expect(condition := rejected, message := 'Recovery rejects missing storage before any child access');
expectDInt(
	expected := -1,
	actual := _MissingConfigurationRunner.ExitCode,
	message := 'Invalid recovery retains abort'
);
rejected := FALSE;

__TRY
	_ExceptionAdsReporter.ReportTestCaseResult(
		groupPath := "",
		testName := "Invalid ADS outcome",
		outcome := TOF_Testing.TEST_OUTCOME.RUNNING,
		duration := T#0S,
		message := diagnostic
	);
__CATCH(exceptionCode)
	assertCaughtExceptionType(exceptionCode := exceptionCode, expectedTypeName := 'ArgumentValueNotSupportedException');
	rejected := TRUE;
__ENDTRY

expect(condition := rejected, message := 'Reporter rejects the actual nonterminal enum value');
checkExceptionClasses := TRUE;
END_METHOD

(*!
<summary>Verifies first-failure summary retention and per-run reset through the ADS reporter callbacks.</summary>
<description>Checks rejected writes, bounded ADS output for a root leaf, and reset on the next run.
Returns TRUE when all observations for this scenario are complete.
</description>
*)
METHOD PRIVATE checkAdsReporterSummary : BOOL
VAR
	diagnostic : TOF_Core.ERROR_MESSAGE;
END_VAR
_AdsSummaryReporter.ReportRunStart(testCount := 2);
_AdsSummaryReporter.RejectWrites := TRUE;
diagnostic := "Synthetic first diagnostic";
_AdsSummaryReporter.ReportTestCaseResult(
	groupPath := "Reporter regression",
	testName := "First leaf",
	outcome := TOF_Testing.TEST_OUTCOME.FAILED,
	duration := T#0S,
	message := diagnostic
);

_AdsSummaryReporter.RejectWrites := FALSE;
diagnostic := "Synthetic second diagnostic";
_AdsSummaryReporter.ReportTestCaseResult(
	groupPath := "Reporter regression",
	testName := "Second leaf",
	outcome := TOF_Testing.TEST_OUTCOME.FAILED,
	duration := T#0S,
	message := diagnostic
);

_AdsSummaryReporter.ReportRunEnd(
	totalTests := 2,
	passedTests := 0,
	failedTests := 2,
	skippedTests := 0,
	duration := T#0S
);

expect(
	condition := _AdsSummaryReporter.LastRunSummary =
		"[TOF_Testing] Finished: 0 passed, 2 failed, 0 skipped | First failure: First leaf: Synthetic first diagnostic",
	message := 'A second failure must preserve the first failure in the summary'
);

expect(
	condition := _AdsSummaryReporter.AcceptedMessage =
		"[TOF_Testing] Finished: 0 passed, 2 failed, 0 skipped | First failed test: First leaf",
	message := 'The completion record must identify the first failure even after its detail write is rejected'
);
expect(
	condition := _AdsSummaryReporter.FailedLogWriteCount = 1,
	message := 'Exactly one rejected write must be counted'
);
expect(
	condition := _AdsSummaryReporter.LastLogFailureMessage =
		"[TOF_Testing] Reporter regression/First leaf: Synthetic first diagnostic",
	message := 'Later accepted writes must preserve the rejected message'
);

_AdsSummaryReporter.ReportRunStart(testCount := 0);

expect(
	condition := _AdsSummaryReporter.LastRunSummary = "",
	message := 'Starting a new run must clear the retained summary'
);
expect(
	condition := _AdsSummaryReporter.FailedLogWriteCount = 0 AND_THEN _AdsSummaryReporter.LastLogFailureMessage = "",
	message := 'A successful start must clear earlier failed-write observations'
);

_AdsSummaryReporter.ReportRunEnd(
	totalTests := 0,
	passedTests := 0,
	failedTests := 0,
	skippedTests := 0,
	duration := T#0S
);

expect(
	condition := _AdsSummaryReporter.LastRunSummary = "[TOF_Testing] Finished: 0 passed, 0 failed, 0 skipped",
	message := 'An empty run must omit the earlier failure'
);

_AdsSummaryReporter.ReportRunStart(testCount := 1);
diagnostic := "Long diagnostic containing a literal %s. ";
TOF_Core.WideStrings.AppendFit255(
	diagnostic,
	"AAAAAAAAAAAAAAAAAAAAAAAAAAAAAAAAAAAAAAAAAAAAAAAAAAAAAAAAAAAAAAAAAAAAAAAAAAAAAAAA",
	"BBBBBBBBBBBBBBBBBBBBBBBBBBBBBBBBBBBBBBBBBBBBBBBBBBBBBBBBBBBBBBBBBBBBBBBBBBBBBBBB",
	"CCCCCCCCCCCCCCCCCCCCCCCCCCCCCCCCCCCCCCCCCCCCCCCCCCCCCCCCCCCCCCCCCCCCCCCCCCCCCCCC"
);
_AdsSummaryReporter.ReportTestCaseResult(
	groupPath := "",
	testName := "Long failure",
	outcome := TOF_Testing.TEST_OUTCOME.FAILED,
	duration := T#0S,
	message := diagnostic
);

expect(
	condition := TOF_Core.WideStrings.GetLength(value := _AdsSummaryReporter.AcceptedMessage) = 200,
	message := 'A long ADS diagnostic must fit within the reporter limit'
);
expect(
	condition := Tc2_Standard.WLEFT(STR := _AdsSummaryReporter.AcceptedMessage, SIZE := 27) =
		"[TOF_Testing] Long failure:",
	message := 'A root leaf is logged without a leading group separator'
);

_AdsSummaryReporter.RejectWrites := TRUE;
_AdsSummaryReporter.ReportRunEnd(
	totalTests := 1,
	passedTests := 0,
	failedTests := 1,
	skippedTests := 0,
	duration := T#0S
);
expect(
	condition := _AdsSummaryReporter.LastLogFailureMessage =
		"[TOF_Testing] Finished: 0 passed, 1 failed, 0 skipped | First failed test: Long failure",
	message := 'Rejection must retain the exact completion record independently of diagnostic length'
);
expect(
	condition := _AdsSummaryReporter.FailedLogWriteCount = 1,
	message := 'A rejected completion record must be counted once'
);
_AdsSummaryReporter.RejectWrites := FALSE;

checkAdsReporterSummary := TRUE;
END_METHOD

(*!
<summary>Recovers a throwing external child, including a failed first recovery attempt.</summary>
<description>Explicitly releases the modeled resource before requesting reset recovery.
Returns TRUE when all observations for this scenario are complete.
</description>
*)
METHOD PRIVATE checkExternalRecovery : BOOL
VAR
	exceptionCode : __SYSTEM.ExceptionCode;
	rejected : BOOL;
	externalCase : REFERENCE TO ExternalElementProbe;
	actualParent : TOF_Testing.ITestElement;
END_VAR
IF NOT _ExternalConfigured THEN
	_ExternalRun.Reporter := _ExternalReport;
	_ExternalConfigured := TRUE;
END_IF

_ExternalRun.Execute(cleanupTaskMemory := FALSE);
_ExternalCalls := _ExternalCalls + 1;

IF NOT _ExternalRun.IsFinished THEN
	IF _ExternalCalls < 16 THEN
		RETURN;
	END_IF

	expect(condition := FALSE, message := 'The external recovery run must finish within 16 scans');
	_ExternalRun.ExternalCase.ReleaseResource();
	checkExternalRecovery := TRUE;

	RETURN;
END_IF

IF NOT _ExternalRecovered THEN
	expectDInt(expected := -1, actual := _ExternalRun.ExitCode, message := 'External child aborts');
	expect(
		condition := _ExternalRun.ExternalCase.ResourceActive,
		message := 'Abort does not silently release user resources'
	);
	_ExternalRun.Execute(cleanupTaskMemory := FALSE);
	expectUDInt(
		expected := 1,
		actual := _ExternalRun.ExternalCase.ExecuteCalls,
		message := 'The aborted callback is not retried before explicit recovery'
	);
	externalCase REF= _ExternalRun.ExternalCase;
	externalCase.ReleaseResource();
	expectFalse(
		condition := externalCase.ResourceActive,
		message := 'Explicit resource release completes before reset recovery'
	);
	externalCase.ThrowOnReset := TRUE;

	__TRY
		_ExternalRun.Reset();
	__CATCH(exceptionCode)
		assertCaughtExceptionType(
			exceptionCode := exceptionCode,
			expectedTypeName := 'StandardException'
		);
		rejected := TRUE;
	__ENDTRY

	expect(condition := rejected, message := 'Custom recovery Reset failure propagates');
	expectDInt(expected := -1, actual := _ExternalRun.ExitCode, message := 'Failed recovery retains abort');
	externalCase.ThrowOnReset := FALSE;
	externalCase.ThrowOnExecute := FALSE;
	_ExternalRun.Reset();
	actualParent := _ExternalRun.ExternalCase.Parent;
	expect(condition := actualParent = 0, message := 'The recovered root remains parentless');
	expectUDInt(
		expected := 3,
		actual := _ExternalRun.ExternalCase.ResetCalls,
		message := 'Failed reset was retried'
	);
	_ExternalRecovered := TRUE;
	_ExternalCalls := 0;
	RETURN;
END_IF

expect(condition := _ExternalRun.AllPassed, message := 'The same static tree succeeds after explicit recovery');
expectDInt(expected := 1, actual := _ExternalRun.PassedTests, message := 'The recovered root contributes one leaf');
expect(condition := _ExternalReport.IsReady, message := 'The recovered run completes its report');
expectUDInt(
	expected := 2,
	actual := _ExternalRun.ExternalCase.ExecuteCalls,
	message := 'Execute resumes only in the new run'
);
checkExternalRecovery := TRUE;
END_METHOD

(*!
<summary>Checks direct-child interface dispatch, fixed ordering and explicit accessor failures.</summary>
<description>
Borrows persistent fixtures before execution and after a rejected Reset. Test-only slot corruption is restored
before returning. Child identity is compared through ITestElement on both sides; indexed observation
invokes no child body.

Returns TRUE when all observations for this scenario are complete.
</description>
*)
METHOD PRIVATE checkIndexedChildren : BOOL
VAR
	element : TOF_Testing.ITestElement;
	parentElement : TOF_Testing.IParentTestElement;
	child : TOF_Testing.ITestElement;
	expectedChild : TOF_Testing.ITestElement;
	supportsChildren : BOOL;
	exceptionCode : __SYSTEM.ExceptionCode;
	rejected : BOOL;
	firstBodyCalls : UDINT;
END_VAR
element := _IndexedGroup;
supportsChildren := __QUERYINTERFACE(element, parentElement);
expect(condition := supportsChildren, message := 'A group exposes the direct-child capability');

IF NOT supportsChildren THEN
	checkIndexedChildren := TRUE;
	RETURN;
END_IF

firstBodyCalls := _IndexedGroup.First.BodyCalls;
expect(condition := parentElement.ChildCount = 2, message := 'The capability reports the fixed direct count');
expectedChild := _IndexedGroup.First;
child := parentElement.GetChildByIndex(index := 0);
expect(condition := child = expectedChild, message := 'Index zero borrows the first child');
expectedChild := _IndexedGroup.Second;
child := parentElement.GetChildByIndex(index := 1);
expect(condition := child = expectedChild, message := 'The last valid index borrows the last child');

__TRY
	child := parentElement.GetChildByIndex(index := 2);
__CATCH(exceptionCode)
	assertCaughtExceptionType(exceptionCode := exceptionCode, expectedTypeName := 'ArgumentOutOfRangeException');
	rejected := TRUE;
__ENDTRY

expect(condition := rejected, message := 'Index equal to ChildCount is rejected');
rejected := FALSE;

__TRY
	child := parentElement.GetChildByIndex(index := TOF_Core.SignedInt16.MAX_VALUE);
__CATCH(exceptionCode)
	assertCaughtExceptionType(exceptionCode := exceptionCode, expectedTypeName := 'ArgumentOutOfRangeException');
	rejected := TRUE;
__ENDTRY

expect(condition := rejected, message := 'The largest representable index is rejected before indexing');
parentElement := _Runner.Empty;
expect(condition := parentElement.ChildCount = TOF_Core.SignedInt16.ZERO, message := 'An empty group reports zero direct children');
rejected := FALSE;

__TRY
	child := parentElement.GetChildByIndex(index := 0);
__CATCH(exceptionCode)
	assertCaughtExceptionType(exceptionCode := exceptionCode, expectedTypeName := 'ArgumentOutOfRangeException');
	rejected := TRUE;
__ENDTRY

expect(condition := rejected, message := 'A valid empty array has no valid child index');
parentElement := _MissingConfigurationGroup;
rejected := FALSE;

__TRY
	child := parentElement.GetChildByIndex(index := TOF_Core.SignedInt16.MAX_VALUE);
__CATCH(exceptionCode)
	assertCaughtExceptionType(exceptionCode := exceptionCode, expectedTypeName := 'DataMemberNotSpecifiedException');
	rejected := TRUE;
__ENDTRY

expect(condition := rejected, message := 'Missing storage is diagnosed before an invalid index');

// A failed Reset does not prevent observing an existing slot; the missing selected slot remains an error.
_IndexedGroup.Children[1] := 0;
rejected := FALSE;

__TRY
	_IndexedGroup.Reset(reporter := 0);
__CATCH(exceptionCode)
	assertCaughtExceptionType(exceptionCode := exceptionCode, expectedTypeName := 'DataMemberNotSpecifiedException');
	rejected := TRUE;
__ENDTRY

expect(condition := rejected, message := 'The injected missing slot rejects Reset');
parentElement := _IndexedGroup;
expectedChild := _IndexedGroup.First;
child := parentElement.GetChildByIndex(index := 0);
expect(condition := child = expectedChild, message := 'An existing slot can be observed after failed Reset');
rejected := FALSE;

__TRY
	child := parentElement.GetChildByIndex(index := 1);
__CATCH(exceptionCode)
	assertCaughtExceptionType(exceptionCode := exceptionCode, expectedTypeName := 'DataMemberNotSpecifiedException');
	rejected := TRUE;
__ENDTRY

expect(condition := rejected, message := 'A null selected slot is a missing member');
_IndexedGroup.Children[1] := _IndexedGroup.Second;
expectUDInt(
	expected := firstBodyCalls,
	actual := _IndexedGroup.First.BodyCalls,
	message := 'Indexed observation invokes no child body'
);
_IndexedGroup.Reset(reporter := 0);
checkIndexedChildren := TRUE;
END_METHOD

(*!
<summary>Checks live root-to-element paths independently of Reset and reporting.</summary>
<description>
Checks interface dispatch, own-name inclusion, empty names, Unicode, root-prefix truncation and cycles among ancestors.
Synthetic parent-only chains isolate GetPath; they are never registered or executed as group compositions.
The existing nested and repeated-run cases independently check JUnit group paths without the leaf name.

Returns TRUE when all observations for this scenario are complete.
</description>
*)
METHOD PRIVATE checkPaths : BOOL
VAR
	element : TOF_Testing.ITestElement;
	named : TOF_Core.INamed;
	actualPath : WSTRING(255);
	expectedPath : WSTRING(255);
	exceptionCode : __SYSTEM.ExceptionCode;
	rejected : BOOL;
	diagnostic : TOF_Core.ERROR_MESSAGE;
	content : POINTER TO STRING;
	longName : WSTRING(81);
	expectedXmlName : STRING(255);
END_VAR
expectedPath := "AAAAAAAAAAAAAAAAAAAAAAAAAAAAAAAAAAAAAAAAAAAAAAAAAAAAAAAAAAAAAAAAAAAAAAAAAAAAAAAA";
named := _PathLongName;
expect(condition := named.Name = expectedPath, message := 'INamed retains the first 80 name characters');
actualPath := _PathLongName.GetPath();
expect(condition := actualPath = expectedPath, message := 'A root path observes the same bounded name');
longName := "AAAAAAAAAAAAAAAAAAAAAAAAAAAAAAAAAAAAAAAAAAAAAAAAAAAAAAAAAAAAAAAAAAAAAAAAAAAAAAAAB";
_PathReport.ReportRunStart(testCount := 1);
_PathReport.ReportTestCaseResult(
	groupPath := "",
	testName := longName,
	outcome := TOF_Testing.TEST_OUTCOME.PASSED,
	duration := T#0S,
	message := diagnostic
);
_PathReport.ReportRunEnd(totalTests := 1, passedTests := 1, failedTests := 0, skippedTests := 0, duration := T#0S);
content := _PathReport.ContentAddress;
expectedXmlName := TOF_Core.Strings.Concat255('name="', TO_STRING(expectedPath), '"');
expect(condition := _PathReport.IsReady AND_THEN content <> 0, message := 'The bounded-name report completes');

IF content <> 0 THEN
	expect(
		condition := TOF_Core.Strings.Contains(stringToSearchIn := content^, stringToFind := expectedXmlName),
		message := 'Reporter input retains exactly the first 80 name characters'
	);
END_IF

element := _DuplicateGroup;
actualPath := element.GetPath();
expect(condition := actualPath = "Duplicates", message := 'A root path contains its own name');
actualPath := _DuplicateGroup.First.GetPath();
expect(condition := actualPath = "Duplicates/First", message := 'A child path includes its group and own name');
actualPath := _Runner.FailureOuter.Failures.BodyFailure.GetPath();
expect(
	condition := actualPath = "Nested/Failures/Body failure",
	message := 'Ancestor names are ordered from the root'
);
actualPath := _Runner.Pass.GetPath();
expect(condition := actualPath = "", message := 'A nameless root has an empty path');
actualPath := _PathEmpty.GetPath();
expectedPath := "AAAAAAAAAAAAAAAAAAAAAAAAAAAAAAAAAAAAAAAAAAAAAAAAAAAAAAAAAAAAAAAAAAAAAAAAAAAAAAAA";
expect(condition := actualPath = expectedPath, message := 'An empty own name adds no separator');
actualPath := _PathUnicode.GetPath();
expectedPath := "AAAAAAAAAAAAAAAAAAAAAAAAAAAAAAAAAAAAAAAAAAAAAAAAAAAAAAAAAAAAAAAAAAAAAAAAAAAAAAAA/Ω";
expect(condition := actualPath = expectedPath, message := 'Empty ancestors are skipped and Unicode is preserved');
actualPath := _PathFourth.GetPath();
expectedPath := Tc2_Utilities.WCONCAT(
	STR1 := "AAAAAAAAAAAAAAAAAAAAAAAAAAAAAAAAAAAAAAAAAAAAAAAAAAAAAAAAAAAAAAAAAAAAAAAAAAAAAAAA/",
	STR2 := "BBBBBBBBBBBBBBBBBBBBBBBBBBBBBBBBBBBBBBBBBBBBBBBBBBBBBBBBBBBBBBBBBBBBBBBBBBBBBBBB/"
);
expectedPath := Tc2_Utilities.WCONCAT(
	STR1 := expectedPath,
	STR2 := "CCCCCCCCCCCCCCCCCCCCCCCCCCCCCCCCCCCCCCCCCCCCCCCCCCCCCCCCCCCCCCCCCCCCCCCCCCCCCCCC/DDDDDDDDDDD…"
);
expect(condition := actualPath = expectedPath, message := 'Overflow retains the root prefix and final ellipsis');

__TRY
	actualPath := _ParentGroup.Child.GetPath();
__CATCH(exceptionCode)
	assertCaughtExceptionType(exceptionCode := exceptionCode, expectedTypeName := 'StandardException');
	rejected := TRUE;
__ENDTRY

expect(condition := rejected, message := 'A cycle among ancestors is rejected without endless traversal');
actualPath := _ReportPathInner.GetPath();
_PathReport.ReportRunStart(testCount := 1);
_PathReport.ReportTestCaseResult(
	groupPath := actualPath,
	testName := "Leaf",
	outcome := TOF_Testing.TEST_OUTCOME.PASSED,
	duration := T#0S,
	message := diagnostic
);
_PathReport.ReportRunEnd(totalTests := 1, passedTests := 1, failedTests := 0, skippedTests := 0, duration := T#0S);
content := _PathReport.ContentAddress;
expect(condition := _PathReport.IsReady AND_THEN content <> 0, message := 'The deep-path report completes');

IF content <> 0 THEN
	expect(
		condition := TOF_Core.Strings.Contains(
			stringToSearchIn := content^,
			stringToFind := 'name="Leaf" classname="Report root/Middle/Inner"'
		),
		message := 'JUnit preserves all three group ancestors and keeps the leaf name separate'
	);
END_IF

checkPaths := TRUE;
END_METHOD

(*!
<summary>Verifies that a reporter failure aborts once after teardown and clears the reporter reference.</summary>
<description>The same leaf runs with a replacement reporter after a completed abort and Reset.
An incomplete run fails when it reaches the scan limit. Returns TRUE when the scenario has an outcome.
</description>
*)
METHOD PRIVATE checkReporterAbort : BOOL
VAR
	exceptionCode : __SYSTEM.ExceptionCode;
	rejected : BOOL;
	diagnostic : TOF_Core.ERROR_MESSAGE;
	actualParent : TOF_Testing.ITestElement;
END_VAR
IF _AbortRecovered THEN
	_AbortRun.Execute(cleanupTaskMemory := FALSE);
	_AbortCalls := _AbortCalls + 1;

	IF NOT _AbortRun.IsFinished AND_THEN _AbortCalls < 16 THEN
		RETURN;
	END_IF

	expect(condition := _AbortRun.IsFinished, message := 'The recovered reporter run finishes within 16 scans');
	expect(condition := _AbortRun.IsFinished AND_THEN _AbortRun.AllPassed,
		message := 'The same static tree passes after reporter abort');
	expectUDInt(
		expected := 1,
		actual := _AbortRun.AbortCase.BodyCalls,
		message := 'The same root executes once in the new run'
	);
	expectUDInt(expected := 1, actual := _AbortReport.ResultCalls, message := 'Old reporter is not retried');
	checkReporterAbort := TRUE;
	RETURN;
END_IF

IF NOT _AbortConfigured THEN

	__TRY
		_InvalidReport.ReportTestCaseResult(
			groupPath := "",
			testName := "Invalid outcome",
			outcome := TOF_Testing.TEST_OUTCOME.NOT_RUN,
			duration := T#0S,
			message := diagnostic
		);
	__CATCH(exceptionCode)
		assertCaughtExceptionType(
			exceptionCode := exceptionCode,
			expectedTypeName := 'ArgumentValueNotSupportedException'
		);
		rejected := TRUE;
	__ENDTRY

	expect(condition := rejected, message := 'A reporter rejects a nonterminal outcome');
	_AbortRun.Reporter := _AbortReport;
	_AbortConfigured := TRUE;
END_IF

_AbortRun.Execute(cleanupTaskMemory := FALSE);
_AbortCalls := _AbortCalls + 1;

IF NOT _AbortRun.IsFinished THEN
	IF _AbortCalls < 16 THEN
		RETURN;
	END_IF

	expect(condition := FALSE, message := 'Callback abort must terminate within 16 scans');
	checkReporterAbort := TRUE;

	RETURN;
END_IF

IF _AbortPostCalls < 2 THEN
	_AbortPostCalls := _AbortPostCalls + 1;
	RETURN;
END_IF

expectDInt(expected := -1, actual := _AbortRun.ExitCode, message := 'Callback abort has a distinct exit code');
expectUDInt(expected := 1, actual := _AbortReport.ResultCalls, message := 'The callback is never retried');
expectUDInt(
	expected := 1,
	actual := _AbortRun.AbortCase.TeardownCalls,
	message := 'Cleanup precedes result reporting'
);
expect(
	condition := _AbortRun.AbortCase.IsFinished AND_THEN _AbortRun.AbortCase.Reporter = 0,
	message := 'A completed leaf clears its reporter reference even when result delivery throws'
);
expectFalse(condition := _AbortReport.IsReady, message := 'An aborted report remains incomplete');
expect(
	condition := TOF_Core.WideStrings.Contains(stringToSearchIn := _AbortRun.CallbackMessage,
		stringToFind := "Reporter failed"),
	message := 'External callback diagnostic is copied'
);
_AbortRun.Reset();
expect(condition := _AbortRun.CallbackMessage = "", message := 'Reset clears copied callback diagnostic');
actualParent := _AbortRun.AbortCase.Parent;
expect(condition := actualParent = 0, message := 'The same root remains parentless after recovery');
_AbortRun.Reporter := _AbortRecoveryReport;
_AbortRecovered := TRUE;
_AbortCalls := 0;
END_METHOD

(*!
<summary>Checks static root validation, recovery guards and absence of cyclic topology scans.</summary>
<description>Deliberately corrupts test-only slots, restoring them before valid recovery and before execution reaches them.
Returns TRUE when all observations for this scenario are complete.
</description>
*)
METHOD PRIVATE checkRunnerTopology : BOOL
VAR
	exceptionCode : __SYSTEM.ExceptionCode;
	rejected : BOOL;
	runningRoot : REFERENCE TO AssertionIsolationProbe;
	actualParent : TOF_Testing.ITestElement;
END_VAR
IF NOT _RootTopologyConfigured THEN
	_RootTopologyRunner.Reporter := _RootTopologyReport;
	_RootTopologyRunner.RootTopologyFirst.Reset(reporter := 0);
	_RootTopologyRunner.RootTopologyFirst.Execute();
	_RootTopologyRunner.Children[1] := 0;
	_RootTopologyRunner.Execute(cleanupTaskMemory := FALSE);
	expectDInt(expected := -1, actual := _RootTopologyRunner.ExitCode, message := 'A null root aborts startup');
	assertCaughtExceptionType(
		exceptionCode := _RootTopologyRunner.CallbackException,
		expectedTypeName := 'DataMemberNotSpecifiedException'
	);
	expect(
		condition := _RootTopologyRunner.RootTopologyFirst.IsFinished,
		message := 'All direct roots are validated before the first Reset'
	);
	expectFalse(condition := _RootTopologyReport.IsReady, message := 'Invalid startup produces no completed report');
	expect(
		condition := _RootTopologyReport.ContentLength = TOF_Core.UnsignedInt32.ZERO,
		message := 'Invalid startup does not call ReportRunStart'
	);
	rejected := FALSE;

	__TRY
		_RootTopologyRunner.Reset();
	__CATCH(exceptionCode)
		assertCaughtExceptionType(exceptionCode := exceptionCode, expectedTypeName := 'DataMemberNotSpecifiedException');
		rejected := TRUE;
	__ENDTRY

	expect(condition := rejected, message := 'Recovery validates slots before dereferencing an invalid tree');
	expectDInt(
		expected := -1,
		actual := _RootTopologyRunner.ExitCode,
		message := 'Failed recovery retains abort'
	);
	_RootTopologyRunner.Children[1] := _RootTopologyRunner.RootTopologyGroup;
	_RootTopologyRunner.Reset();
	_RootTopologyRunner.Children[1] := _RootTopologyRunner.RootTopologyFirst;
	_RootTopologyRunner.Execute(cleanupTaskMemory := FALSE);
	expectDInt(
		expected := -1,
		actual := _RootTopologyRunner.ExitCode,
		message := 'Duplicate roots abort startup'
	);
	assertCaughtExceptionType(exceptionCode := _RootTopologyRunner.CallbackException, expectedTypeName := 'StandardException');
	_RootTopologyRunner.Children[1] := _RootTopologyRunner.RootTopologyGroup;
	_RootTopologyRunner.Reset();
	_RootTopologyRunner.Children[0] := _RootTopologyRunner.RootTopologyGroup.Child;
	_RootTopologyRunner.Execute(cleanupTaskMemory := FALSE);
	expectDInt(
		expected := -1,
		actual := _RootTopologyRunner.ExitCode,
		message := 'A group-owned root aborts startup'
	);
	assertCaughtExceptionType(exceptionCode := _RootTopologyRunner.CallbackException, expectedTypeName := 'StandardException');
	_RootTopologyRunner.Children[0] := _RootTopologyRunner.RootTopologyFirst;
	_RootTopologyRunner.Reset();
	_RootTopologyRunner.RootTopologyFirst.Execute();
	_RootTopologyRunner.Children[1] := _Runner.FailureOuter.Failures;
	_RootTopologyRunner.Execute(cleanupTaskMemory := FALSE);
	expectDInt(
		expected := -1,
		actual := _RootTopologyRunner.ExitCode,
		message := 'A nested group cannot also occupy a root slot'
	);
	assertCaughtExceptionType(exceptionCode := _RootTopologyRunner.CallbackException, expectedTypeName := 'StandardException');
	expect(
		condition := _RootTopologyRunner.RootTopologyFirst.IsFinished,
		message := 'Owned-group rejection occurs before the first direct Reset'
	);
	expect(
		condition := _RootTopologyReport.ContentLength = TOF_Core.UnsignedInt32.ZERO,
		message := 'Owned-group rejection does not start reporting'
	);
	rejected := FALSE;

	__TRY
		_RootTopologyRunner.Reset();
	__CATCH(exceptionCode)
		assertCaughtExceptionType(exceptionCode := exceptionCode, expectedTypeName := 'StandardException');
		rejected := TRUE;
	__ENDTRY

	expect(condition := rejected, message := 'Abort recovery also rejects a group-owned root');
	expectDInt(expected := -1, actual := _RootTopologyRunner.ExitCode, message := 'Invalid recovery retains abort');
	_RootTopologyRunner.Children[1] := _RootTopologyRunner.RootTopologyGroup;
	_RootTopologyRunner.Reset();
	runningRoot REF= _RootTopologyRunner.RunningRoot;
	runningRoot.Timeout := T#0S;
	_RootTopologyRunner.RunningRoot.Reset(reporter := 0);
	_RootTopologyRunner.RunningRoot.Execute();
	expect(condition := _RootTopologyRunner.RunningRoot.IsRunning, message := 'The active-root fixture is pending');
	_RootTopologyRunner.Children[0] := _RootTopologyRunner.RunningRoot;
	_RootTopologyRunner.Execute(cleanupTaskMemory := FALSE);
	expectDInt(
		expected := -1,
		actual := _RootTopologyRunner.ExitCode,
		message := 'An active root aborts startup'
	);
	assertCaughtExceptionType(exceptionCode := _RootTopologyRunner.CallbackException, expectedTypeName := 'StandardException');
	_RootTopologyRunner.RunningRoot.Reset(reporter := 0);
	_RootTopologyRunner.Children[0] := _RootTopologyRunner.RootTopologyFirst;
	_RootTopologyRunner.Reset();
	_RootTopologyRunner.Execute(cleanupTaskMemory := FALSE);
	expectFalse(condition := _RootTopologyRunner.IsFinished, message := 'Valid startup prepares the static roots');

	// Fault injection: restore the unused slot immediately after driving the first root.
	_RootTopologyRunner.Children[1] := 0;
	_RootTopologyRunner.Execute(cleanupTaskMemory := FALSE);
	_RootTopologyRunner.Children[1] := _RootTopologyRunner.RootTopologyGroup;
	expectDInt(
		expected := 0,
		actual := _RootTopologyRunner.ExitCode,
		message := 'Execution does not rescan root slots'
	);
	_RootTopologyConfigured := TRUE;
END_IF

_RootTopologyRunner.Execute(cleanupTaskMemory := FALSE);
_RootTopologyCalls := _RootTopologyCalls + 1;

IF NOT _RootTopologyRunner.IsFinished AND_THEN _RootTopologyCalls < 16 THEN
	RETURN;
END_IF

expect(condition := _RootTopologyRunner.IsFinished, message := 'The topology run finishes within 16 scans');
expect(
	condition := _RootTopologyRunner.IsFinished AND_THEN _RootTopologyRunner.AllPassed,
	message := 'The owned static roots execute successfully'
);
expectDInt(
	expected := 2,
	actual := _RootTopologyRunner.PassedTests,
	message := 'Two direct or nested leaves pass'
);
expectUDInt(
	expected := 1,
	actual := _RootTopologyRunner.RootTopologyFirst.BodyCalls,
	message := 'The first root executes once in the valid run'
);
expectUDInt(
	expected := 1,
	actual := _RootTopologyRunner.RootTopologyGroup.Child.BodyCalls,
	message := 'The nested group executes its owned leaf'
);
actualParent := _RootTopologyRunner.RootTopologyFirst.Parent;
expect(condition := actualParent = 0, message := 'Runner roots remain parentless');
actualParent := _RootTopologyRunner.RootTopologyGroup.Child.Parent;
expect(
	condition := actualParent <> 0,
	message := 'A nested leaf retains its constructor-assigned parent'
);
checkRunnerTopology := TRUE;
END_METHOD

(*!
<summary>Checks fixed parents, missing or repeated children, parent mismatch, cycles, ordered dispatch and repeat execution.</summary>
<description>
Fault injection deliberately mutates a test-only array between rejected operations and briefly during execution
to detect redundant validation. Restore every unused slot before execution reaches it.

Returns TRUE when all observations for this scenario are complete.
</description>
*)
METHOD PRIVATE checkTopology : BOOL
VAR
	exceptionCode : __SYSTEM.ExceptionCode;
	rejected : BOOL;
	expectedParent : TOF_Testing.ITestElement;
	actualParent : TOF_Testing.ITestElement;
END_VAR
expectedParent := _DuplicateGroup;
actualParent := _DuplicateGroup.First.Parent;
expect(condition := actualParent = expectedParent, message := 'Parent is assigned at construction');
actualParent := _DuplicateGroup.Parent;
expect(condition := actualParent = 0, message := 'A root is constructed without a parent');

// Deliberately corrupt the borrowed test-only array to inject topology faults.
// A later execution probe restores its unused slot before that slot is reached.
_DuplicateGroup.Children[1] := 0;

__TRY
	_DuplicateGroup.Reset(reporter := 0);
__CATCH(exceptionCode)
	assertCaughtExceptionType(exceptionCode := exceptionCode, expectedTypeName := 'DataMemberNotSpecifiedException');
	rejected := TRUE;
__ENDTRY

expect(condition := rejected, message := 'A null fixed child is rejected by Reset');
expectUDInt(
	expected := 0,
	actual := _DuplicateGroup.First.BodyCalls,
	message := 'No earlier child body executes'
);
rejected := FALSE;
_DuplicateGroup.Children[1] := _DuplicateGroup.First;

__TRY
	_DuplicateGroup.Reset(reporter := 0);
__CATCH(exceptionCode)
	assertCaughtExceptionType(exceptionCode := exceptionCode, expectedTypeName := 'StandardException');
	rejected := TRUE;
__ENDTRY

expect(condition := rejected, message := 'Duplicate fixed slots are rejected');
rejected := FALSE;
_DuplicateGroup.Children[1] := _RootTopologyRunner.RootTopologyGroup.Child;

__TRY
	_DuplicateGroup.Reset(reporter := 0);
__CATCH(exceptionCode)
	assertCaughtExceptionType(exceptionCode := exceptionCode, expectedTypeName := 'StandardException');
	rejected := TRUE;
__ENDTRY

expect(condition := rejected, message := 'A child assigned to another group is rejected');
actualParent := _DuplicateGroup.First.Parent;
expect(condition := actualParent = expectedParent, message := 'Rejection never changes Parent');
_DuplicateGroup.Children[1] := _DuplicateGroup.Second;
rejected := FALSE;

__TRY
	_ParentGroup.Reset(reporter := 0);
__CATCH(exceptionCode)
	assertCaughtExceptionType(exceptionCode := exceptionCode, expectedTypeName := 'StandardException');
	rejected := TRUE;
__ENDTRY

expect(condition := rejected, message := 'A cycle assigned by constructors is rejected before recursion');

_DuplicateGroup.Reset(reporter := 0);
// Fault injection: an unused slot must not be rescanned in Execute; restore before that slot is reached.
_DuplicateGroup.Children[1] := 0;
_DuplicateGroup.Execute();
expectUDInt(
	expected := 1,
	actual := _DuplicateGroup.First.BodyCalls,
	message := 'The first Execute reaches the first owned child through Children'
);
expectUDInt(
	expected := 0,
	actual := _DuplicateGroup.Second.BodyCalls,
	message := 'The first Execute does not reach the second owned child'
);
_DuplicateGroup.Children[1] := _DuplicateGroup.Second;
_DuplicateGroup.Execute();
expect(condition := _DuplicateGroup.IsFinished, message := 'A valid static group finishes without Configure');
expectDInt(expected := 2, actual := _DuplicateGroup.PassedCount, message := 'Both owned leaves pass');
_DuplicateGroup.Reset(reporter := 0);
_DuplicateGroup.Execute();
_DuplicateGroup.Execute();
expectDInt(
	expected := 2,
	actual := _DuplicateGroup.PassedCount,
	message := 'Reset supports another fixed-tree run'
);
expectUDInt(
	expected := 1,
	actual := _DuplicateGroup.First.BodyCalls,
	message := 'A repeated leaf executes once'
);
actualParent := _DuplicateGroup.First.Parent;
expect(condition := actualParent = expectedParent, message := 'Repeated runs preserve Parent');
_DuplicateGroup.Children[1] := 0;
rejected := FALSE;

__TRY
	_DuplicateGroup.Reset(reporter := 0);
__CATCH(exceptionCode)
	assertCaughtExceptionType(exceptionCode := exceptionCode, expectedTypeName := 'DataMemberNotSpecifiedException');
	rejected := TRUE;
__ENDTRY

expect(condition := rejected, message := 'Invalid topology is rejected on a later Reset too');
expect(
	condition := _DuplicateGroup.First.IsFinished,
	message := 'Validation precedes the first direct child Reset'
);
_DuplicateGroup.Children[1] := _DuplicateGroup.Second;
checkTopology := TRUE;
END_METHOD

(*!
<summary>Checks long XML diagnostics, supplementary Unicode, isolated surrogates and XML controls.</summary>
<description>Returns TRUE when all observations for this scenario are complete.</description>
*)
METHOD PRIVATE checkXmlEncoding : BOOL
VAR
	diagnostic : TOF_Core.ERROR_MESSAGE;
	characters : POINTER TO WORD;
	content : POINTER TO STRING;
	i : UDINT;
END_VAR
// U+1F600 is a surrogate pair; it is followed by an isolated high surrogate, U+0001, TAB and ampersand.
characters := ADR(diagnostic);
characters[0] := 16#D83D;
characters[1] := 16#DE00;
characters[2] := 16#D800;
characters[3] := 16#0001;
characters[4] := 16#0009;
characters[5] := 16#0026;

FOR i := 6 TO 405 DO
	characters[i] := 16#0078;
END_FOR

characters[406] := TOF_Core.UnsignedInt16.MIN_VALUE;
TOF_Core.WideStrings.AppendFit(targetString := diagnostic, sourceString := "END_OF_XML_DIAGNOSTIC");
_XmlReport.ReportRunStart(testCount := 1);
_XmlReport.ReportTestCaseResult(
	groupPath := "Wide",
	testName := "",
	outcome := TOF_Testing.TEST_OUTCOME.FAILED,
	duration := T#1250MS,
	message := diagnostic
);
_XmlReport.ReportRunEnd(totalTests := 1, passedTests := 0, failedTests := 1, skippedTests := 0, duration := T#1250MS);
content := _XmlReport.ContentAddress;
expect(condition := _XmlReport.IsReady AND_THEN content <> 0, message := 'Completed Unicode XML has a buffer');

IF content <> 0 THEN
	expect(
		condition := TOF_Core.Strings.Contains(stringToSearchIn := content^,
			stringToFind := '&#128512;&#65533;&#65533;&#9;&amp;'),
		message := 'Surrogate pair, isolated surrogate, forbidden control and tab are encoded'
	);
	expect(
		condition := TOF_Core.Strings.Contains(stringToSearchIn := content^, stringToFind := 'END_OF_XML_DIAGNOSTIC'),
		message := 'Diagnostic suffix beyond 255 characters survives'
	);
	expect(
		condition := TOF_Core.Strings.Contains(stringToSearchIn := content^, stringToFind := 'time="1.250"'),
		message := 'JUnit duration uses decimal seconds'
	);
END_IF

checkXmlEncoding := TRUE;
END_METHOD

(*!
<summary>Repeats a nested run and checks configured and completed leaf counts, cleanup and escaped JUnit output.</summary>
<description>Configures owned fixtures through borrowed references without copying their state.
Returns TRUE when all observations for this scenario are complete.
</description>
*)
METHOD PRIVATE runAndCheck : BOOL
VAR
	content : POINTER TO STRING;
	probe : REFERENCE TO TestingProbe;
	multiCycleProbe : REFERENCE TO AssertionIsolationProbe;
END_VAR
IF NOT _Configured THEN
	expectDInt(expected := 5, actual := _Runner.FailureOuter.TestCount, message := 'Nested leaf count');
	expectDInt(expected := 0, actual := _Runner.Empty.TestCount, message := 'Empty group leaf count');
	expectDInt(expected := 1, actual := _Runner.Pass.TestCount, message := 'Single-cycle leaf count');
	expectDInt(expected := 1, actual := _Runner.Multi.TestCount, message := 'Multi-cycle leaf count');

	probe REF= _Runner.FailureOuter.Failures.SetupFailure;
	probe.ThrowBeforeTest := TRUE;
	probe REF= _Runner.FailureOuter.Failures.BodyFailure;
	probe.ThrowBody := TRUE;
	probe REF= _Runner.FailureOuter.Failures.TeardownFailure;
	probe.ThrowAfterTest := TRUE;
	probe REF= _Runner.FailureOuter.Failures.ComparisonFailure;
	probe.InvalidComparison := TRUE;
	probe REF= _Runner.FailureOuter.Failures.DiagnosticFailure;
	probe.DiagnosticFailure := TRUE;
	_Runner.Reporter := _Reporter;
	multiCycleProbe REF= _Runner.Multi;
	multiCycleProbe.Timeout := T#0S;
	_Configured := TRUE;
END_IF

_Runner.Execute(cleanupTaskMemory := FALSE);
_Calls := _Calls + 1;

IF NOT _Runner.IsFinished AND_THEN _Calls < 32 THEN
	RETURN;
END_IF

expect(condition := _Runner.IsFinished, message := 'The tree finishes within 32 scans');
expectDInt(expected := 2, actual := _Runner.PassedTests, message := 'Single and multi-cycle leaves pass');
expectDInt(expected := 5, actual := _Runner.FailedTests, message := 'Five distinct leaf failures');
expectDInt(expected := 7, actual := _Runner.TotalTests, message := 'Groups add no synthetic tests');
expectDInt(expected := 5, actual := _Runner.FailureOuter.TestCount, message := 'Leaf count survives a run');
expectUDInt(
	expected := 0,
	actual := _Runner.FailureOuter.Failures.SetupFailure.BodyCalls,
	message := 'Failed setup suppresses body'
);
expectUDInt(
	expected := 1,
	actual := _Runner.FailureOuter.Failures.SetupFailure.TeardownCalls,
	message := 'Failed setup still cleans up'
);
expectUDInt(
	expected := 1,
	actual := _Runner.FailureOuter.Failures.BodyFailure.TeardownCalls,
	message := 'Thrown body cleans up'
);
expectUDInt(
	expected := 1,
	actual := _Runner.FailureOuter.Failures.TeardownFailure.TeardownCalls,
	message := 'Thrown teardown is not retried'
);
expectUDInt(
	expected := 1,
	actual := _Runner.Pass.BodyCalls,
	message := 'Single-cycle body executes once per run'
);
expectUDInt(
	expected := 3,
	actual := _Runner.Multi.BodyCalls,
	message := 'Multi-cycle state survives three scans'
);
expectDInt(
	expected := 0,
	actual := _Runner.Empty.FailedCount,
	message := 'An empty group passes without tests'
);
expect(condition := _Reporter.IsReady, message := 'JUnit output is complete');
expect(
	condition := TOF_Core.WideStrings.Contains(stringToSearchIn := _Runner.FailureOuter.Failures.SetupFailure.FailureMessage,
		stringToFind := "BeforeTest: "),
	message := 'Preparation stage survives exception capture'
);
expect(
	condition := TOF_Core.WideStrings.Contains(stringToSearchIn := _Runner.FailureOuter.Failures.BodyFailure.FailureMessage,
		stringToFind := "Body failed"),
	message := 'Framework payload survives task cleanup'
);
expect(
	condition := TOF_Core.WideStrings.Contains(stringToSearchIn := _Runner.FailureOuter.Failures.BodyFailure.FailureMessage,
		stringToFind := "ExecuteTest"),
	message := 'Framework source survives task cleanup'
);
expect(
	condition := TOF_Core.WideStrings.Contains(stringToSearchIn := _Runner.FailureOuter.Failures.TeardownFailure.FailureMessage,
		stringToFind := "Teardown failed"),
	message := 'Teardown payload is copied'
);

content := _Reporter.ContentAddress;
expect(condition := content <> 0, message := 'Completed XML exposes a buffer');

IF content <> 0 THEN
	expect(
		condition := TOF_Core.Strings.Contains(
			stringToSearchIn := content^,
			stringToFind := 'Expected value &lt; '
		),
		message := 'An incompatible borrowed comparison remains an assertion failure'
	);
	expect(
		condition := TOF_Core.Strings.Contains(stringToSearchIn := content^, stringToFind := '&#1070;&amp;&lt;'),
		message := 'Cyrillic and XML markup are preserved'
	);
	expect(
		condition := TOF_Core.Strings.Contains(stringToSearchIn := content^, stringToFind := 'name=""'),
		message := 'Empty test name serializes safely'
	);
	expect(
		condition := TOF_Core.Strings.Contains(stringToSearchIn := content^, stringToFind := 'classname="Nested/Failures"'),
		message := 'The nested group path is preserved'
	);
END_IF

IF NOT _Repeated AND_THEN _Runner.IsFinished THEN
	_Repeated := TRUE;
	_Calls := 0;
	_Runner.Reset();
	RETURN;
END_IF

runAndCheck := TRUE;
END_METHOD

(*!
<summary>Borrows the initialized concrete class name.</summary>
*)
{attribute 'monitoring' := 'call'}
PROPERTY ClassName : REFERENCE TO STRING
GET
ClassName REF= _ClassName;
END_GET
END_PROPERTY

(*!
<summary>Borrows the project namespace name.</summary>
*)
{attribute 'monitoring' := 'call'}
PROPERTY NamespaceName : REFERENCE TO STRING
GET
NamespaceName REF= CurrentNamespace.Name;
END_GET
END_PROPERTY

END_FUNCTION_BLOCK

// ---- Tests/Testing/MixedTestRunner.TcPOU
(*
SPDX-License-Identifier: MIT
License: https://opensource.org/license/mit
*)

(*!
<summary>Runs mixed outcomes, nested groups, an empty group and a multi-cycle test.</summary>
<description>
Owns persistent root instances and fixed child storage. Use from one task without reentry.
Children borrows the same array for the instance lifetime. Root parents remain zero.
Instances must not be copied because their fixtures contain non-copyable state.
</description>
*)

{attribute 'no_assign'}
{attribute 'no_explicit_call' := 'do not call this function block directly'}
FUNCTION_BLOCK MixedTestRunner EXTENDS TOF_Testing.TestRunner<4>
VAR_STAT
	//! <summary>Class name shared by instances of this concrete runner.</summary>
	{attribute 'hide'}
	_ClassName : STRING := __POUNAME();
END_VAR
VAR_OUTPUT
	//! <summary>Owned root element used by this runner.</summary>
	FailureOuter : NestedFailureTestGroup(name := "Nested", parent := 0);
	//! <summary>Owned root element used by this runner.</summary>
	Empty : EmptyTestGroup(name := "Empty", parent := 0);
	//! <summary>Owned root element used by this runner.</summary>
	Pass : TestingProbe(name := "", parent := 0);
	//! <summary>Owned root element used by this runner.</summary>
	Multi : AssertionIsolationProbe(name := "Three cycles", parent := 0);
END_VAR
VAR
	_Children : ARRAY [0.._ChildCount - 1] OF TOF_Testing.ITestElement :=
	[
		FailureOuter,
		Pass,
		Multi,
		Empty
	];
END_VAR

(*!
<summary>Borrows the unchanged persistent root array; application code must not modify it.</summary>
*)
{attribute 'monitoring' := 'call'}
PROPERTY Children : REFERENCE TO ARRAY [0.._ChildCount - 1] OF TOF_Testing.ITestElement
GET
Children REF= _Children;
END_GET
END_PROPERTY

(*!
<summary>Borrows the concrete class name; callers must not modify the returned storage.</summary>
*)
{attribute 'monitoring' := 'call'}
PROPERTY ClassName : REFERENCE TO STRING
GET
ClassName REF= _ClassName;
END_GET
END_PROPERTY

(*!
<summary>Borrows the test project namespace; callers must not modify the returned storage.</summary>
*)
{attribute 'monitoring' := 'call'}
PROPERTY NamespaceName : REFERENCE TO STRING
GET
NamespaceName REF= CurrentNamespace.Name;
END_GET
END_PROPERTY

(*!
<summary>Reports the complete concrete instance size.</summary>
*)
{attribute 'monitoring' := 'call'}
PROPERTY SelfSize : ULINT
GET
SelfSize := XSIZEOF(THIS^);
END_GET
END_PROPERTY

END_FUNCTION_BLOCK

// ---- Tests/Testing/NestedFailureTestGroup.TcPOU
(*
SPDX-License-Identifier: MIT
License: https://opensource.org/license/mit
*)

(*!
<summary>Owns a nested group of failure scenarios.</summary>
<description>
Owns persistent child storage and fixed parent associations. Use in one task without reentry.
Children is borrowed and must not be modified by application code. Constructor callbacks are not used.
</description>
*)

{attribute 'no_assign'}
{attribute 'no_explicit_call' := 'do not call this function block directly'}
FUNCTION_BLOCK NestedFailureTestGroup EXTENDS TOF_Testing.TestGroup<1>
VAR_STAT
	//! <summary>Class name shared by all instances of this function block.</summary>
	{attribute 'hide'}
	_ClassName : STRING := __POUNAME();
END_VAR
VAR
	{attribute 'hide'}
	{attribute 'init_namespace'}
	_NamespaceName : STRING;
END_VAR
VAR_OUTPUT
	//! <summary>Owned nested failure group.</summary>
	Failures : FailureTestGroup(name := "Failures", parent := THIS^);
END_VAR
VAR
	_Children : ARRAY [0.._ChildCount - 1] OF TOF_Testing.ITestElement :=
	[
		Failures
	];
END_VAR

//! <summary>Borrows the concrete class name for the lifetime of this instance; callers must not modify it.</summary>
{attribute 'monitoring' := 'call'}
PROPERTY ClassName : REFERENCE TO STRING
GET
ClassName REF= _ClassName;
END_GET
END_PROPERTY

//! <summary>Borrows the compiler-initialized namespace; callers must not modify the returned reference.</summary>
{attribute 'monitoring' := 'call'}
PROPERTY NamespaceName : REFERENCE TO STRING
GET
NamespaceName REF= _NamespaceName;
END_GET
END_PROPERTY

//! <summary>Reports the complete concrete instance size, excluding separately allocated storage.</summary>
{attribute 'monitoring' := 'call'}
PROPERTY SelfSize : ULINT
GET
SelfSize := XSIZEOF(THIS^);
END_GET
END_PROPERTY

//! <summary>Borrows the fixed array of this concrete group; do not modify it.</summary>
{attribute 'monitoring' := 'call'}
PROPERTY Children : REFERENCE TO ARRAY [0.._ChildCount - 1] OF TOF_Testing.ITestElement
GET
Children REF= _Children;
END_GET
END_PROPERTY

END_FUNCTION_BLOCK

// ---- Tests/Testing/FailureTestGroup.TcPOU
(*
SPDX-License-Identifier: MIT
License: https://opensource.org/license/mit
*)

(*!
<summary>Owns the five independent failure scenarios used by the runner suite.</summary>
<description>
Owns persistent child storage and fixed parent associations. Use in one task without reentry.
Children is borrowed and must not be modified by application code. Constructor callbacks are not used.
</description>
*)

{attribute 'no_assign'}
{attribute 'no_explicit_call' := 'do not call this function block directly'}
FUNCTION_BLOCK FailureTestGroup EXTENDS TOF_Testing.TestGroup<5>
VAR_STAT
	//! <summary>Class name shared by all instances of this function block.</summary>
	{attribute 'hide'}
	_ClassName : STRING := __POUNAME();
END_VAR
VAR
	{attribute 'hide'}
	{attribute 'init_namespace'}
	_NamespaceName : STRING;
END_VAR
VAR_OUTPUT
	//! <summary>Leaf configured to raise from preparation.</summary>
	SetupFailure : TestingProbe(name := "Setup failure", parent := THIS^);
	//! <summary>Leaf configured to raise from its body.</summary>
	BodyFailure : TestingProbe(name := "Body failure", parent := THIS^);
	//! <summary>Leaf configured to raise from teardown.</summary>
	TeardownFailure : TestingProbe(name := "Teardown failure", parent := THIS^);
	//! <summary>Leaf configured to record an incompatible-comparison failure.</summary>
	ComparisonFailure : TestingProbe(name := "Comparison failure", parent := THIS^);
	//! <summary>Leaf configured to retain a Unicode diagnostic.</summary>
	DiagnosticFailure : TestingProbe(name := "Diagnostic failure", parent := THIS^);
END_VAR
VAR
	_Children : ARRAY [0.._ChildCount - 1] OF TOF_Testing.ITestElement :=
	[
		SetupFailure,
		BodyFailure,
		TeardownFailure,
		ComparisonFailure,
		DiagnosticFailure
	];
END_VAR

//! <summary>Borrows the concrete class name for the lifetime of this instance; callers must not modify it.</summary>
{attribute 'monitoring' := 'call'}
PROPERTY ClassName : REFERENCE TO STRING
GET
ClassName REF= _ClassName;
END_GET
END_PROPERTY

//! <summary>Borrows the compiler-initialized namespace; callers must not modify the returned reference.</summary>
{attribute 'monitoring' := 'call'}
PROPERTY NamespaceName : REFERENCE TO STRING
GET
NamespaceName REF= _NamespaceName;
END_GET
END_PROPERTY

//! <summary>Reports the complete concrete instance size, excluding separately allocated storage.</summary>
{attribute 'monitoring' := 'call'}
PROPERTY SelfSize : ULINT
GET
SelfSize := XSIZEOF(THIS^);
END_GET
END_PROPERTY

//! <summary>Borrows the fixed array of this concrete group; do not modify it.</summary>
{attribute 'monitoring' := 'call'}
PROPERTY Children : REFERENCE TO ARRAY [0.._ChildCount - 1] OF TOF_Testing.ITestElement
GET
Children REF= _Children;
END_GET
END_PROPERTY

END_FUNCTION_BLOCK

// ---- Tests/Testing/TestingProbe.TcPOU
(*
SPDX-FileCopyrightText: © 2026 Oleksandr Tiutyk <trofimich@gmail.com>
SPDX-License-Identifier: MIT
License: https://opensource.org/license/mit
*)

(*!
<summary>Provides one configurable single-cycle scenario for runner regression tests.</summary>
<description>
Persistent fixture state owns its exception template. BeforeTest resets per-run observations.
</description>
*)

{attribute 'no_explicit_call' := 'do not call this function block directly'}
FUNCTION_BLOCK TestingProbe EXTENDS TOF_Testing.SingleCycleTest
VAR_INPUT
	ThrowBeforeTest : BOOL;
	ThrowBody : BOOL;
	ThrowAfterTest : BOOL;
	InvalidComparison : BOOL;
	DiagnosticFailure : BOOL;
END_VAR
VAR_OUTPUT
	SetupCalls : UDINT;
	BodyCalls : UDINT;
	TeardownCalls : UDINT;
END_VAR
VAR
	_Exception : TOF_Core.StandardException;
END_VAR
VAR_STAT
	//! <summary>Class name shared by all instances of this function block.</summary>
	{attribute 'hide'}
	_ClassName : STRING := __POUNAME();
END_VAR
VAR
	{attribute 'hide'}
	{attribute 'init_namespace'}
	_NamespaceName : STRING;
END_VAR

(*!
<summary>Resets observations and optionally raises during scenario preparation.</summary>
*)
METHOD PROTECTED BeforeTest
SetupCalls := 1;
BodyCalls := 0;
TeardownCalls := 0;

IF ThrowBeforeTest THEN
	_Exception.Throw(
		sourceNamespaceName := NamespaceName,
		sourceClassName := ClassName,
		sourcePOUName := __POUNAME(),
		sourcePosition := __POSITION(),
		message := "Setup failed"
	);
END_IF
END_METHOD

(*!
<summary>Runs one successful body or one selected failure route.</summary>
*)
METHOD PROTECTED ExecuteTest
VAR
	textValue : STRING(255);
	integerValue : DINT;
END_VAR
BodyCalls := BodyCalls + 1;

IF ThrowBody THEN
	_Exception.Throw(
		sourceNamespaceName := NamespaceName,
		sourceClassName := ClassName,
		sourcePOUName := __POUNAME(),
		sourcePosition := __POSITION(),
		message := "Body failed"
	);
END_IF

IF InvalidComparison THEN
	textValue := 'text';
	integerValue := 1;
	Assert.That(actual := textValue).IsLessThan(expected := integerValue);
ELSIF DiagnosticFailure THEN
	RecordFailure(message := "$042E&<");
ELSE
	Assert.ThatDInt(actual := 2 + 3).ToBe(expected := 5);
END_IF
END_METHOD

(*!
<summary>Counts cleanup exactly once and optionally raises after its side effect.</summary>
*)
METHOD PROTECTED AfterTest
TeardownCalls := TeardownCalls + 1;

IF ThrowAfterTest THEN
	_Exception.Throw(
		sourceNamespaceName := NamespaceName,
		sourceClassName := ClassName,
		sourcePOUName := __POUNAME(),
		sourcePosition := __POSITION(),
		message := "Teardown failed"
	);
END_IF
END_METHOD

//! <summary>Borrows the concrete class name for the lifetime of this instance; callers must not modify it.</summary>
{attribute 'monitoring' := 'call'}
PROPERTY ClassName : REFERENCE TO STRING
GET
ClassName REF= _ClassName;
END_GET
END_PROPERTY

//! <summary>Borrows the compiler-initialized namespace; callers must not modify the returned reference.</summary>
{attribute 'monitoring' := 'call'}
PROPERTY NamespaceName : REFERENCE TO STRING
GET
NamespaceName REF= _NamespaceName;
END_GET
END_PROPERTY

//! <summary>Reports the complete concrete instance size, excluding separately allocated storage.</summary>
{attribute 'monitoring' := 'call'}
PROPERTY SelfSize : ULINT
GET
SelfSize := XSIZEOF(THIS^);
END_GET
END_PROPERTY

END_FUNCTION_BLOCK

// ---- Tests/Testing/EmptyTestGroup.TcPOU
(*
SPDX-License-Identifier: MIT
License: https://opensource.org/license/mit
*)

(*!
<summary>Provides a concrete group with an empty child array.</summary>
<description>
Owns persistent child storage and fixed parent associations. Use in one task without reentry.
Children is borrowed and must not be modified by application code. Constructor callbacks are not used.
</description>
*)

{attribute 'no_assign'}
{attribute 'no_explicit_call' := 'do not call this function block directly'}
FUNCTION_BLOCK EmptyTestGroup EXTENDS TOF_Testing.TestGroup<0>
VAR_STAT
	//! <summary>Class name shared by all instances of this function block.</summary>
	{attribute 'hide'}
	_ClassName : STRING := __POUNAME();
END_VAR
VAR
	_Children : ARRAY [0.._ChildCount - 1] OF TOF_Testing.ITestElement;
END_VAR

//! <summary>Borrows the concrete class name for the lifetime of this instance; callers must not modify it.</summary>
{attribute 'monitoring' := 'call'}
PROPERTY ClassName : REFERENCE TO STRING
GET
ClassName REF= _ClassName;
END_GET
END_PROPERTY

//! <summary>Borrows the test project namespace; callers must not modify the returned reference.</summary>
{attribute 'monitoring' := 'call'}
PROPERTY NamespaceName : REFERENCE TO STRING
GET
NamespaceName REF= CurrentNamespace.Name;
END_GET
END_PROPERTY

//! <summary>Reports the complete concrete instance size, excluding separately allocated storage.</summary>
{attribute 'monitoring' := 'call'}
PROPERTY SelfSize : ULINT
GET
SelfSize := XSIZEOF(THIS^);
END_GET
END_PROPERTY

//! <summary>Borrows the fixed array of this concrete group; do not modify it.</summary>
{attribute 'monitoring' := 'call'}
PROPERTY Children : REFERENCE TO ARRAY [0.._ChildCount - 1] OF TOF_Testing.ITestElement
GET
Children REF= _Children;
END_GET
END_PROPERTY

END_FUNCTION_BLOCK

// ---- Tests/Testing/AssertionIsolationProbe.TcPOU
(*
SPDX-FileCopyrightText: © 2026 Oleksandr Tiutyk <trofimich@gmail.com>
SPDX-License-Identifier: MIT
License: https://opensource.org/license/mit
*)

(*!
<summary>Exercises bounded multi-cycle completion and case-owned failure routing.</summary>
<description>
A nonzero Peer is failed during this body. Zero CompleteAfterCycle leaves completion to the deadline.
FailSelfWhileBusy asserts FALSE while returning TEST_CYCLE_RESULT.BUSY to verify immediate failure termination.
</description>
*)

{attribute 'no_explicit_call' := 'do not call this function block directly'}
FUNCTION_BLOCK AssertionIsolationProbe EXTENDS TOF_Testing.MultiCycleTest
VAR_INPUT
	Peer : POINTER TO AssertionIsolationProbe;
	UseDirectFailure : BOOL;
	FailSelfWhileBusy : BOOL;
	CompleteAfterCycle : UDINT := 3;
END_VAR
VAR_OUTPUT
	BodyCalls : UDINT;
	TeardownCalls : UDINT;
END_VAR
VAR_STAT
	//! <summary>Class name shared by all instances of this function block.</summary>
	{attribute 'hide'}
	_ClassName : STRING := __POUNAME();
END_VAR
VAR
	{attribute 'hide'}
	{attribute 'init_namespace'}
	_NamespaceName : STRING;
END_VAR

(*!
<summary>Resets per-run fixture observations.</summary>
*)
METHOD PROTECTED BeforeTest
BodyCalls := 0;
TeardownCalls := 0;
END_METHOD

(*!
<summary>Waits across scans or fails a peer and returns whether the scenario is done.</summary>
*)
METHOD PROTECTED ExecuteTest : TOF_Testing.TEST_CYCLE_RESULT
BodyCalls := BodyCalls + 1;

IF FailSelfWhileBusy THEN
	Assert.ThatBool(actual := FALSE).IsTrue();
	ExecuteTest := TOF_Testing.TEST_CYCLE_RESULT.BUSY;
ELSIF Peer <> 0 THEN
	Peer^.FailActiveCase(useDirectFailure := UseDirectFailure);
	ExecuteTest := TOF_Testing.TEST_CYCLE_RESULT.DONE;
ELSIF CompleteAfterCycle > TOF_Core.UnsignedInt32.ZERO AND_THEN CycleCount >= CompleteAfterCycle THEN
	Assert.ThatUDInt(actual := BodyCalls).ToBe(expected := CompleteAfterCycle);
	ExecuteTest := TOF_Testing.TEST_CYCLE_RESULT.DONE;
ELSE
	ExecuteTest := TOF_Testing.TEST_CYCLE_RESULT.BUSY;
END_IF
END_METHOD

(*!
<summary>Counts one cleanup for success, peer failure or timeout.</summary>
*)
METHOD PROTECTED AfterTest
TeardownCalls := TeardownCalls + 1;
END_METHOD

(*!
<summary>Reports through the receiving case while a different case is executing.</summary>
*)
METHOD INTERNAL FailActiveCase
VAR_INPUT
	useDirectFailure : BOOL;
END_VAR
IF useDirectFailure THEN
	RecordFailure(message := "Failure belongs to this case");
ELSE
	Assert.ThatBool(actual := FALSE).IsTrue();
END_IF
END_METHOD

//! <summary>Borrows the concrete class name for the lifetime of this instance; callers must not modify it.</summary>
{attribute 'monitoring' := 'call'}
PROPERTY ClassName : REFERENCE TO STRING
GET
ClassName REF= _ClassName;
END_GET
END_PROPERTY

//! <summary>Borrows the compiler-initialized namespace; callers must not modify the returned reference.</summary>
{attribute 'monitoring' := 'call'}
PROPERTY NamespaceName : REFERENCE TO STRING
GET
NamespaceName REF= _NamespaceName;
END_GET
END_PROPERTY

//! <summary>Reports the complete concrete instance size, excluding separately allocated storage.</summary>
{attribute 'monitoring' := 'call'}
PROPERTY SelfSize : ULINT
GET
SelfSize := XSIZEOF(THIS^);
END_GET
END_PROPERTY

END_FUNCTION_BLOCK

// ---- Tests/Testing/IsolationTestRunner.TcPOU
(*
SPDX-License-Identifier: MIT
License: https://opensource.org/license/mit
*)

(*!
<summary>Runs one owned multi-cycle probe for independent assertion routing.</summary>
<description>
Owns persistent root instances and fixed child storage. Use from one task without reentry.
Children borrows the same array for the instance lifetime. Root parents remain zero.
</description>
*)

{attribute 'no_assign'}
{attribute 'no_explicit_call' := 'do not call this function block directly'}
FUNCTION_BLOCK IsolationTestRunner EXTENDS TOF_Testing.TestRunner<1>
VAR_STAT
	//! <summary>Class name shared by instances of this concrete runner.</summary>
	{attribute 'hide'}
	_ClassName : STRING := __POUNAME();
END_VAR
VAR
	{attribute 'hide'}
	{attribute 'init_namespace'}
	_NamespaceName : STRING;
END_VAR
VAR_OUTPUT
	//! <summary>Owned root element used by this runner.</summary>
	Child : AssertionIsolationProbe(name := "Receiver", parent := 0);
END_VAR
VAR
	_Children : ARRAY [0.._ChildCount - 1] OF TOF_Testing.ITestElement :=
	[
		Child
	];
END_VAR

(*!
<summary>Borrows the concrete class name; callers must not modify the returned storage.</summary>
*)
{attribute 'monitoring' := 'call'}
PROPERTY ClassName : REFERENCE TO STRING
GET
ClassName REF= _ClassName;
END_GET
END_PROPERTY

(*!
<summary>Borrows the concrete namespace name for the instance lifetime; callers must not modify it.</summary>
*)
{attribute 'monitoring' := 'call'}
PROPERTY NamespaceName : REFERENCE TO STRING
GET
NamespaceName REF= _NamespaceName;
END_GET
END_PROPERTY

(*!
<summary>Reports the complete concrete instance size.</summary>
*)
{attribute 'monitoring' := 'call'}
PROPERTY SelfSize : ULINT
GET
SelfSize := XSIZEOF(THIS^);
END_GET
END_PROPERTY

(*!
<summary>Borrows the unchanged persistent root array; application code must not modify it.</summary>
*)
{attribute 'monitoring' := 'call'}
PROPERTY Children : REFERENCE TO ARRAY [0.._ChildCount - 1] OF TOF_Testing.ITestElement
GET
Children REF= _Children;
END_GET
END_PROPERTY

END_FUNCTION_BLOCK

// ---- Tests/Testing/AssertionCallerTestRunner.TcPOU
(*
SPDX-License-Identifier: MIT
License: https://opensource.org/license/mit
*)

(*!
<summary>Runs the owned caller that reports a failure to another active case.</summary>
<description>
Owns persistent root instances and fixed child storage. Use from one task without reentry.
Children borrows the same array for the instance lifetime. Root parents remain zero.
</description>
*)

{attribute 'no_assign'}
{attribute 'no_explicit_call' := 'do not call this function block directly'}
FUNCTION_BLOCK AssertionCallerTestRunner EXTENDS TOF_Testing.TestRunner<1>
VAR_STAT
	//! <summary>Class name shared by instances of this concrete runner.</summary>
	{attribute 'hide'}
	_ClassName : STRING := __POUNAME();
END_VAR
VAR
	{attribute 'hide'}
	{attribute 'init_namespace'}
	_NamespaceName : STRING;
END_VAR
VAR_OUTPUT
	//! <summary>Owned root element used by this runner.</summary>
	Child : AssertionIsolationProbe(name := "Caller", parent := 0);
END_VAR
VAR
	_Children : ARRAY [0.._ChildCount - 1] OF TOF_Testing.ITestElement :=
	[
		Child
	];
END_VAR

(*!
<summary>Borrows the concrete class name; callers must not modify the returned storage.</summary>
*)
{attribute 'monitoring' := 'call'}
PROPERTY ClassName : REFERENCE TO STRING
GET
ClassName REF= _ClassName;
END_GET
END_PROPERTY

(*!
<summary>Borrows the concrete namespace name for the instance lifetime; callers must not modify it.</summary>
*)
{attribute 'monitoring' := 'call'}
PROPERTY NamespaceName : REFERENCE TO STRING
GET
NamespaceName REF= _NamespaceName;
END_GET
END_PROPERTY

(*!
<summary>Reports the complete concrete instance size.</summary>
*)
{attribute 'monitoring' := 'call'}
PROPERTY SelfSize : ULINT
GET
SelfSize := XSIZEOF(THIS^);
END_GET
END_PROPERTY

(*!
<summary>Borrows the unchanged persistent root array; application code must not modify it.</summary>
*)
{attribute 'monitoring' := 'call'}
PROPERTY Children : REFERENCE TO ARRAY [0.._ChildCount - 1] OF TOF_Testing.ITestElement
GET
Children REF= _Children;
END_GET
END_PROPERTY

END_FUNCTION_BLOCK

// ---- Tests/Testing/EmptyTestRunner.TcPOU
(*
SPDX-License-Identifier: MIT
License: https://opensource.org/license/mit
*)

(*!
<summary>Runs a valid empty root array without synthetic test results.</summary>
<description>
Owns persistent root instances and fixed child storage. Use from one task without reentry.
Children borrows the same array for the instance lifetime. Root parents remain zero.
</description>
*)

{attribute 'no_assign'}
{attribute 'no_explicit_call' := 'do not call this function block directly'}
FUNCTION_BLOCK EmptyTestRunner EXTENDS TOF_Testing.TestRunner<0>
VAR_STAT
	//! <summary>Class name shared by instances of this concrete runner.</summary>
	{attribute 'hide'}
	_ClassName : STRING := __POUNAME();
END_VAR
VAR
	{attribute 'hide'}
	{attribute 'init_namespace'}
	_NamespaceName : STRING;
END_VAR
VAR
	_Children : ARRAY [0.._ChildCount - 1] OF TOF_Testing.ITestElement;
END_VAR

(*!
<summary>Borrows the concrete class name; callers must not modify the returned storage.</summary>
*)
{attribute 'monitoring' := 'call'}
PROPERTY ClassName : REFERENCE TO STRING
GET
ClassName REF= _ClassName;
END_GET
END_PROPERTY

(*!
<summary>Borrows the concrete namespace name for the instance lifetime; callers must not modify it.</summary>
*)
{attribute 'monitoring' := 'call'}
PROPERTY NamespaceName : REFERENCE TO STRING
GET
NamespaceName REF= _NamespaceName;
END_GET
END_PROPERTY

(*!
<summary>Reports the complete concrete instance size.</summary>
*)
{attribute 'monitoring' := 'call'}
PROPERTY SelfSize : ULINT
GET
SelfSize := XSIZEOF(THIS^);
END_GET
END_PROPERTY

(*!
<summary>Borrows the unchanged persistent root array; application code must not modify it.</summary>
*)
{attribute 'monitoring' := 'call'}
PROPERTY Children : REFERENCE TO ARRAY [0.._ChildCount - 1] OF TOF_Testing.ITestElement
GET
Children REF= _Children;
END_GET
END_PROPERTY

END_FUNCTION_BLOCK

// ---- Tests/Testing/ReporterAbortTestRunner.TcPOU
(*
SPDX-License-Identifier: MIT
License: https://opensource.org/license/mit
*)

(*!
<summary>Runs one owned leaf for reporter abort and restart regressions.</summary>
<description>
Owns persistent root instances and fixed child storage. Use from one task without reentry.
Children borrows the same array for the instance lifetime. Root parents remain zero.
</description>
*)

{attribute 'no_assign'}
{attribute 'no_explicit_call' := 'do not call this function block directly'}
FUNCTION_BLOCK ReporterAbortTestRunner EXTENDS TOF_Testing.TestRunner<1>
VAR_STAT
	//! <summary>Class name shared by instances of this concrete runner.</summary>
	{attribute 'hide'}
	_ClassName : STRING := __POUNAME();
END_VAR
VAR
	{attribute 'hide'}
	{attribute 'init_namespace'}
	_NamespaceName : STRING;
END_VAR
VAR_OUTPUT
	//! <summary>Owned root element used by this runner.</summary>
	AbortCase : TestingProbe(name := "Reporter abort", parent := 0);
END_VAR
VAR
	_Children : ARRAY [0.._ChildCount - 1] OF TOF_Testing.ITestElement :=
	[
		AbortCase
	];
END_VAR

(*!
<summary>Borrows the concrete class name; callers must not modify the returned storage.</summary>
*)
{attribute 'monitoring' := 'call'}
PROPERTY ClassName : REFERENCE TO STRING
GET
ClassName REF= _ClassName;
END_GET
END_PROPERTY

(*!
<summary>Borrows the concrete namespace name for the instance lifetime; callers must not modify it.</summary>
*)
{attribute 'monitoring' := 'call'}
PROPERTY NamespaceName : REFERENCE TO STRING
GET
NamespaceName REF= _NamespaceName;
END_GET
END_PROPERTY

(*!
<summary>Reports the complete concrete instance size.</summary>
*)
{attribute 'monitoring' := 'call'}
PROPERTY SelfSize : ULINT
GET
SelfSize := XSIZEOF(THIS^);
END_GET
END_PROPERTY

(*!
<summary>Borrows the unchanged persistent root array; application code must not modify it.</summary>
*)
{attribute 'monitoring' := 'call'}
PROPERTY Children : REFERENCE TO ARRAY [0.._ChildCount - 1] OF TOF_Testing.ITestElement
GET
Children REF= _Children;
END_GET
END_PROPERTY

END_FUNCTION_BLOCK

// ---- Tests/Testing/ThrowingTestReporter.TcPOU
(*
SPDX-FileCopyrightText: © 2026 Oleksandr Tiutyk <trofimich@gmail.com>
SPDX-License-Identifier: MIT
License: https://opensource.org/license/mit
*)

(*!
<summary>Raises after observing a leaf callback to verify abort without callback retries.</summary>
*)

{attribute 'no_explicit_call' := 'do not call this function block directly'}
FUNCTION_BLOCK ThrowingTestReporter EXTENDS TOF_Testing.JUnitXmlReporter
VAR_STAT
	_ThrowingClassName : STRING := __POUNAME();
END_VAR
VAR_OUTPUT
	ResultCalls : UDINT;
END_VAR
VAR
	_Exception : TOF_Core.StandardException;
END_VAR

(*!
<summary>Counts a side effect and raises from the external reporter callback.</summary>
<param name="testName">Individual name bounded to 80 wide characters, matching the reporter interface.</param>
*)
METHOD ReportTestCaseResult
VAR_INPUT
	groupPath : WSTRING(255);
	testName : WSTRING;
	outcome : TOF_Testing.TEST_OUTCOME;
	duration : TIME;
END_VAR
VAR_IN_OUT CONSTANT
	message : TOF_Core.ERROR_MESSAGE;
END_VAR
ResultCalls := ResultCalls + 1;
_Exception.Throw(
	sourceNamespaceName := NamespaceName,
	sourceClassName := ClassName,
	sourcePOUName := __POUNAME(),
	sourcePosition := __POSITION(),
	message := "Reporter failed"
);
END_METHOD

//! <summary>Provides concrete reporter fixture metadata.</summary>
{attribute 'monitoring' := 'call'}
PROPERTY ClassName : REFERENCE TO STRING
GET
ClassName REF= _ThrowingClassName;
END_GET
END_PROPERTY

//! <summary>Reports this concrete fixture size.</summary>
{attribute 'monitoring' := 'call'}
PROPERTY SelfSize : ULINT
GET
SelfSize := XSIZEOF(THIS^);
END_GET
END_PROPERTY

END_FUNCTION_BLOCK

// ---- Tests/Testing/DeadlineTestRunner.TcPOU
(*
SPDX-License-Identifier: MIT
License: https://opensource.org/license/mit
*)

(*!
<summary>Runs an owned group containing a test controlled by its deadline.</summary>
<description>
Owns persistent root instances and fixed child storage. Use from one task without reentry.
Children borrows the same array for the instance lifetime. Root parents remain zero.
</description>
*)

{attribute 'no_assign'}
{attribute 'no_explicit_call' := 'do not call this function block directly'}
FUNCTION_BLOCK DeadlineTestRunner EXTENDS TOF_Testing.TestRunner<1>
VAR_STAT
	//! <summary>Class name shared by instances of this concrete runner.</summary>
	{attribute 'hide'}
	_ClassName : STRING := __POUNAME();
END_VAR
VAR
	{attribute 'hide'}
	{attribute 'init_namespace'}
	_NamespaceName : STRING;
END_VAR
VAR_OUTPUT
	//! <summary>Owned root element used by this runner.</summary>
	DeadlineGroup : DeadlineTestGroup(name := "Deadline group", parent := 0);
END_VAR
VAR
	_Children : ARRAY [0.._ChildCount - 1] OF TOF_Testing.ITestElement :=
	[
		DeadlineGroup
	];
END_VAR

(*!
<summary>Borrows the concrete class name; callers must not modify the returned storage.</summary>
*)
{attribute 'monitoring' := 'call'}
PROPERTY ClassName : REFERENCE TO STRING
GET
ClassName REF= _ClassName;
END_GET
END_PROPERTY

(*!
<summary>Borrows the concrete namespace name for the instance lifetime; callers must not modify it.</summary>
*)
{attribute 'monitoring' := 'call'}
PROPERTY NamespaceName : REFERENCE TO STRING
GET
NamespaceName REF= _NamespaceName;
END_GET
END_PROPERTY

(*!
<summary>Reports the complete concrete instance size.</summary>
*)
{attribute 'monitoring' := 'call'}
PROPERTY SelfSize : ULINT
GET
SelfSize := XSIZEOF(THIS^);
END_GET
END_PROPERTY

(*!
<summary>Borrows the unchanged persistent root array; application code must not modify it.</summary>
*)
{attribute 'monitoring' := 'call'}
PROPERTY Children : REFERENCE TO ARRAY [0.._ChildCount - 1] OF TOF_Testing.ITestElement
GET
Children REF= _Children;
END_GET
END_PROPERTY

END_FUNCTION_BLOCK

// ---- Tests/Testing/DeadlineTestGroup.TcPOU
(*
SPDX-License-Identifier: MIT
License: https://opensource.org/license/mit
*)

(*!
<summary>Owns the pending multi-cycle test used for deadline verification.</summary>
<description>
Owns persistent child storage and fixed parent associations. Use in one task without reentry.
Children is borrowed and must not be modified by application code. Constructor callbacks are not used.
</description>
*)

{attribute 'no_assign'}
{attribute 'no_explicit_call' := 'do not call this function block directly'}
FUNCTION_BLOCK DeadlineTestGroup EXTENDS TOF_Testing.TestGroup<1>
VAR_STAT
	//! <summary>Class name shared by all instances of this function block.</summary>
	{attribute 'hide'}
	_ClassName : STRING := __POUNAME();
END_VAR
VAR
	{attribute 'hide'}
	{attribute 'init_namespace'}
	_NamespaceName : STRING;
END_VAR
VAR_OUTPUT
	//! <summary>Owned multi-cycle leaf with an externally selected deadline.</summary>
	Child : AssertionIsolationProbe(name := "Deadline", parent := THIS^);
END_VAR
VAR
	_Children : ARRAY [0.._ChildCount - 1] OF TOF_Testing.ITestElement :=
	[
		Child
	];
END_VAR

//! <summary>Borrows the concrete class name for the lifetime of this instance; callers must not modify it.</summary>
{attribute 'monitoring' := 'call'}
PROPERTY ClassName : REFERENCE TO STRING
GET
ClassName REF= _ClassName;
END_GET
END_PROPERTY

//! <summary>Borrows the compiler-initialized namespace; callers must not modify the returned reference.</summary>
{attribute 'monitoring' := 'call'}
PROPERTY NamespaceName : REFERENCE TO STRING
GET
NamespaceName REF= _NamespaceName;
END_GET
END_PROPERTY

//! <summary>Reports the complete concrete instance size, excluding separately allocated storage.</summary>
{attribute 'monitoring' := 'call'}
PROPERTY SelfSize : ULINT
GET
SelfSize := XSIZEOF(THIS^);
END_GET
END_PROPERTY

//! <summary>Borrows the fixed array of this concrete group; do not modify it.</summary>
{attribute 'monitoring' := 'call'}
PROPERTY Children : REFERENCE TO ARRAY [0.._ChildCount - 1] OF TOF_Testing.ITestElement
GET
Children REF= _Children;
END_GET
END_PROPERTY

END_FUNCTION_BLOCK

// ---- Tests/Testing/PairTestGroup.TcPOU
(*
SPDX-License-Identifier: MIT
License: https://opensource.org/license/mit
*)

(*!
<summary>Owns two ordered single-cycle tests for topology regressions.</summary>
<description>
Owns persistent child storage and fixed parent associations. Use in one task without reentry.
Children is borrowed and must not be modified by application code. Constructor callbacks are not used.
Regression tests may deliberately corrupt the exposed array between failed operations to inject topology faults.
</description>
*)

{attribute 'no_assign'}
{attribute 'no_explicit_call' := 'do not call this function block directly'}
FUNCTION_BLOCK PairTestGroup EXTENDS TOF_Testing.TestGroup<2>
VAR_STAT
	//! <summary>Class name shared by all instances of this function block.</summary>
	{attribute 'hide'}
	_ClassName : STRING := __POUNAME();
END_VAR
VAR
	{attribute 'hide'}
	{attribute 'init_namespace'}
	_NamespaceName : STRING;
END_VAR
VAR_OUTPUT
	//! <summary>First owned regression leaf.</summary>
	First : TestingProbe(name := "First", parent := THIS^);
	//! <summary>Second owned regression leaf.</summary>
	Second : TestingProbe(name := "Second", parent := THIS^);
END_VAR
VAR
	_Children : ARRAY [0.._ChildCount - 1] OF TOF_Testing.ITestElement :=
	[
		First,
		Second
	];
END_VAR

//! <summary>Borrows the concrete class name for the lifetime of this instance; callers must not modify it.</summary>
{attribute 'monitoring' := 'call'}
PROPERTY ClassName : REFERENCE TO STRING
GET
ClassName REF= _ClassName;
END_GET
END_PROPERTY

//! <summary>Borrows the compiler-initialized namespace; callers must not modify the returned reference.</summary>
{attribute 'monitoring' := 'call'}
PROPERTY NamespaceName : REFERENCE TO STRING
GET
NamespaceName REF= _NamespaceName;
END_GET
END_PROPERTY

//! <summary>Reports the complete concrete instance size, excluding separately allocated storage.</summary>
{attribute 'monitoring' := 'call'}
PROPERTY SelfSize : ULINT
GET
SelfSize := XSIZEOF(THIS^);
END_GET
END_PROPERTY

//! <summary>Borrows the fixed array of this concrete group; do not modify it.</summary>
{attribute 'monitoring' := 'call'}
PROPERTY Children : REFERENCE TO ARRAY [0.._ChildCount - 1] OF TOF_Testing.ITestElement
GET
Children REF= _Children;
END_GET
END_PROPERTY

END_FUNCTION_BLOCK

// ---- Tests/Testing/SingleChildTestGroup.TcPOU
(*
SPDX-License-Identifier: MIT
License: https://opensource.org/license/mit
*)

(*!
<summary>Owns one single-cycle regression test.</summary>
<description>
Owns persistent child storage and fixed parent associations. Use in one task without reentry.
Children is borrowed and must not be modified by application code. Constructor callbacks are not used.
</description>
*)

{attribute 'no_assign'}
{attribute 'no_explicit_call' := 'do not call this function block directly'}
FUNCTION_BLOCK SingleChildTestGroup EXTENDS TOF_Testing.TestGroup<1>
VAR_STAT
	//! <summary>Class name shared by all instances of this function block.</summary>
	{attribute 'hide'}
	_ClassName : STRING := __POUNAME();
END_VAR
VAR
	{attribute 'hide'}
	{attribute 'init_namespace'}
	_NamespaceName : STRING;
END_VAR
VAR_OUTPUT
	//! <summary>Owned leaf exposed for regression observations and scenario selection.</summary>
	Child : TestingProbe(name := "Owned leaf", parent := THIS^);
END_VAR
VAR
	_Children : ARRAY [0.._ChildCount - 1] OF TOF_Testing.ITestElement :=
	[
		Child
	];
END_VAR

//! <summary>Borrows the concrete class name for the lifetime of this instance; callers must not modify it.</summary>
{attribute 'monitoring' := 'call'}
PROPERTY ClassName : REFERENCE TO STRING
GET
ClassName REF= _ClassName;
END_GET
END_PROPERTY

//! <summary>Borrows the compiler-initialized namespace; callers must not modify the returned reference.</summary>
{attribute 'monitoring' := 'call'}
PROPERTY NamespaceName : REFERENCE TO STRING
GET
NamespaceName REF= _NamespaceName;
END_GET
END_PROPERTY

//! <summary>Reports the complete concrete instance size, excluding separately allocated storage.</summary>
{attribute 'monitoring' := 'call'}
PROPERTY SelfSize : ULINT
GET
SelfSize := XSIZEOF(THIS^);
END_GET
END_PROPERTY

//! <summary>Borrows the fixed array of this concrete group; do not modify it.</summary>
{attribute 'monitoring' := 'call'}
PROPERTY Children : REFERENCE TO ARRAY [0.._ChildCount - 1] OF TOF_Testing.ITestElement
GET
Children REF= _Children;
END_GET
END_PROPERTY

END_FUNCTION_BLOCK

// ---- Tests/Testing/ExternalRecoveryTestRunner.TcPOU
(*
SPDX-License-Identifier: MIT
License: https://opensource.org/license/mit
*)

(*!
<summary>Runs an owned external element with explicit abort recovery.</summary>
<description>
Owns persistent root instances and fixed child storage. Use from one task without reentry.
Children borrows the same array for the instance lifetime. Root parents remain zero.
</description>
*)

{attribute 'no_assign'}
{attribute 'no_explicit_call' := 'do not call this function block directly'}
FUNCTION_BLOCK ExternalRecoveryTestRunner EXTENDS TOF_Testing.TestRunner<1>
VAR_STAT
	//! <summary>Class name shared by instances of this concrete runner.</summary>
	{attribute 'hide'}
	_ClassName : STRING := __POUNAME();
END_VAR
VAR
	{attribute 'hide'}
	{attribute 'init_namespace'}
	_NamespaceName : STRING;
END_VAR
VAR_OUTPUT
	//! <summary>Owned root element used by this runner.</summary>
	ExternalCase : ExternalElementProbe(name := "External element", parent := 0);
END_VAR
VAR
	_Children : ARRAY [0.._ChildCount - 1] OF TOF_Testing.ITestElement :=
	[
		ExternalCase
	];
END_VAR

(*!
<summary>Borrows the concrete class name; callers must not modify the returned storage.</summary>
*)
{attribute 'monitoring' := 'call'}
PROPERTY ClassName : REFERENCE TO STRING
GET
ClassName REF= _ClassName;
END_GET
END_PROPERTY

(*!
<summary>Borrows the concrete namespace name for the instance lifetime; callers must not modify it.</summary>
*)
{attribute 'monitoring' := 'call'}
PROPERTY NamespaceName : REFERENCE TO STRING
GET
NamespaceName REF= _NamespaceName;
END_GET
END_PROPERTY

(*!
<summary>Reports the complete concrete instance size.</summary>
*)
{attribute 'monitoring' := 'call'}
PROPERTY SelfSize : ULINT
GET
SelfSize := XSIZEOF(THIS^);
END_GET
END_PROPERTY

(*!
<summary>Borrows the unchanged persistent root array; application code must not modify it.</summary>
*)
{attribute 'monitoring' := 'call'}
PROPERTY Children : REFERENCE TO ARRAY [0.._ChildCount - 1] OF TOF_Testing.ITestElement
GET
Children REF= _Children;
END_GET
END_PROPERTY

END_FUNCTION_BLOCK

// ---- Tests/Testing/ExternalElementProbe.TcPOU
(*
SPDX-FileCopyrightText: © 2026 Oleksandr Tiutyk <trofimich@gmail.com>
SPDX-License-Identifier: MIT
License: https://opensource.org/license/mit
*)

(*!
<summary>Exercises external element abort and retryable reset recovery.</summary>
<description>
ResourceActive models a user resource and must be cleared through ReleaseResource before recovery.
Reset never releases it or retries Execute. Disable ThrowOnExecute before a successful subsequent run.
No allocation or I/O is performed.
Use from the hosting test task only.
</description>
*)

{attribute 'no_explicit_call' := 'do not call this function block directly'}
FUNCTION_BLOCK ExternalElementProbe EXTENDS TOF_Testing.TestElement
VAR_INPUT
	//! <summary>Raises from Execute until the recovery test explicitly enables a successful new run.</summary>
	ThrowOnExecute : BOOL := TRUE;
	ThrowOnReset : BOOL;
END_VAR
VAR_OUTPUT
	//! <summary>Whether the modeled resource still requires explicit ReleaseResource before recovery.</summary>
	ResourceActive : BOOL;
	ExecuteCalls : UDINT;
	ResetCalls : UDINT;
END_VAR
VAR
	_Exception : TOF_Core.StandardException;
END_VAR
VAR_STAT
	//! <summary>Class name shared by all instances of this function block.</summary>
	{attribute 'hide'}
	_ClassName : STRING := __POUNAME();
END_VAR
VAR
	{attribute 'hide'}
	{attribute 'init_namespace'}
	_NamespaceName : STRING;
END_VAR

(*!
<summary>Raises with a modeled resource or completes a subsequent explicitly recovered run.</summary>
<description>
When ThrowOnExecute is FALSE, completes one passing result without acquiring the modeled resource.
The borrowed reporter receives that result once with the live parent path; path-provider and reporter failures propagate.
A completed element ignores Execute until Reset.
</description>
*)
METHOD Execute
VAR
	groupPath : WSTRING(255);
	diagnostic : TOF_Core.ERROR_MESSAGE;
END_VAR
IF IsFinished THEN
	RETURN;
END_IF

_State := TOF_Testing.TEST_ELEMENT_STATE.RUNNING;
ExecuteCalls := ExecuteCalls + 1;

IF ThrowOnExecute THEN
	ResourceActive := TRUE;
	_Exception.Throw(
		sourceNamespaceName := NamespaceName,
		sourceClassName := ClassName,
		sourcePOUName := __POUNAME(),
		sourcePosition := __POSITION(),
		message := "External element failed"
	);
END_IF

_PassedCount := 1;
_State := TOF_Testing.TEST_ELEMENT_STATE.COMPLETED;

IF _Reporter <> 0 THEN
	IF _Parent <> 0 THEN
		groupPath := _Parent.GetPath();
	END_IF

	_Reporter.ReportTestCaseResult(
		groupPath := groupPath,
		testName := _Name,
		outcome := TOF_Testing.TEST_OUTCOME.PASSED,
		duration := T#0S,
		message := diagnostic
	);
END_IF

_Reporter := 0;
END_METHOD

(*!
<summary>Releases the resource modeled by this regression fixture.</summary>
<description>
Clears ResourceActive without changing execution state, callback counters or failure controls.
Repeated calls are a no-op. Performs no allocation or I/O and raises no exception. Use from the hosting test task.
</description>
*)
METHOD ReleaseResource
ResourceActive := FALSE;
END_METHOD

(*!
<summary>Counts reset attempts and optionally fails without releasing the modeled resource.</summary>
<description>
Failure occurs before common observations are reset. A subsequent explicit Reset can retry the same operation.
Successful reset delegates common state and reporter binding to the base without releasing ResourceActive.
</description>
<param name="reporter">Borrowed reporter for the next run, or zero to suppress reporting.</param>
*)
METHOD Reset
VAR_INPUT
	reporter : TOF_Testing.ITestReporter;
END_VAR
ResetCalls := ResetCalls + 1;

IF ThrowOnReset THEN
	_Exception.Throw(
		sourceNamespaceName := NamespaceName,
		sourceClassName := ClassName,
		sourcePOUName := __POUNAME(),
		sourcePosition := __POSITION(),
		message := "External reset failed"
	);
END_IF

SUPER^.Reset(reporter := reporter);
END_METHOD

//! <summary>Borrows the concrete class name for the lifetime of this instance; callers must not modify it.</summary>
{attribute 'monitoring' := 'call'}
PROPERTY ClassName : REFERENCE TO STRING
GET
ClassName REF= _ClassName;
END_GET
END_PROPERTY

//! <summary>Borrows the compiler-initialized namespace; callers must not modify the returned reference.</summary>
{attribute 'monitoring' := 'call'}
PROPERTY NamespaceName : REFERENCE TO STRING
GET
NamespaceName REF= _NamespaceName;
END_GET
END_PROPERTY

//! <summary>Reports the complete concrete instance size, excluding separately allocated storage.</summary>
{attribute 'monitoring' := 'call'}
PROPERTY SelfSize : ULINT
GET
SelfSize := XSIZEOF(THIS^);
END_GET
END_PROPERTY

(*!
<summary>Counts the single scenario represented by this fixture.</summary>
*)
{attribute 'monitoring' := 'call'}
PROPERTY TestCount : TOF_Core.DINT_LENGTH
GET
TestCount := 1;
END_GET
END_PROPERTY

END_FUNCTION_BLOCK

// ---- Tests/Testing/DiagnosticTestRunner.TcPOU
(*
SPDX-License-Identifier: MIT
License: https://opensource.org/license/mit
*)

(*!
<summary>Runs native, formatter and long-message diagnostic probes.</summary>
<description>
Owns persistent root instances and fixed child storage. Use from one task without reentry.
Children borrows the same array for the instance lifetime. Root parents remain zero.
</description>
*)

{attribute 'no_assign'}
{attribute 'no_explicit_call' := 'do not call this function block directly'}
FUNCTION_BLOCK DiagnosticTestRunner EXTENDS TOF_Testing.TestRunner<3>
VAR_STAT
	//! <summary>Class name shared by instances of this concrete runner.</summary>
	{attribute 'hide'}
	_ClassName : STRING := __POUNAME();
END_VAR
VAR
	{attribute 'hide'}
	{attribute 'init_namespace'}
	_NamespaceName : STRING;
END_VAR
VAR_OUTPUT
	//! <summary>Owned root element used by this runner.</summary>
	NativeDiagnostic : DiagnosticProbe(name := "Native diagnostic", parent := 0);
	//! <summary>Owned root element used by this runner.</summary>
	FormatterDiagnostic : DiagnosticProbe(name := "Formatter diagnostic", parent := 0);
	//! <summary>Owned root element used by this runner.</summary>
	LongDiagnostic : DiagnosticProbe(name := "Long diagnostic", parent := 0);
END_VAR
VAR
	_Children : ARRAY [0.._ChildCount - 1] OF TOF_Testing.ITestElement :=
	[
		NativeDiagnostic,
		FormatterDiagnostic,
		LongDiagnostic
	];
END_VAR

(*!
<summary>Borrows the concrete class name; callers must not modify the returned storage.</summary>
*)
{attribute 'monitoring' := 'call'}
PROPERTY ClassName : REFERENCE TO STRING
GET
ClassName REF= _ClassName;
END_GET
END_PROPERTY

(*!
<summary>Borrows the concrete namespace name for the instance lifetime; callers must not modify it.</summary>
*)
{attribute 'monitoring' := 'call'}
PROPERTY NamespaceName : REFERENCE TO STRING
GET
NamespaceName REF= _NamespaceName;
END_GET
END_PROPERTY

(*!
<summary>Reports the complete concrete instance size.</summary>
*)
{attribute 'monitoring' := 'call'}
PROPERTY SelfSize : ULINT
GET
SelfSize := XSIZEOF(THIS^);
END_GET
END_PROPERTY

(*!
<summary>Borrows the unchanged persistent root array; application code must not modify it.</summary>
*)
{attribute 'monitoring' := 'call'}
PROPERTY Children : REFERENCE TO ARRAY [0.._ChildCount - 1] OF TOF_Testing.ITestElement
GET
Children REF= _Children;
END_GET
END_PROPERTY

END_FUNCTION_BLOCK

// ---- Tests/Testing/DiagnosticProbe.TcPOU
(*
SPDX-FileCopyrightText: © 2026 Oleksandr Tiutyk <trofimich@gmail.com>
SPDX-License-Identifier: MIT
License: https://opensource.org/license/mit
*)

(*!
<summary>Exercises native errors, failing exception formatting and long copied diagnostics.</summary>
<description>
The existing ThrowingGetMessageException fixture preserves its concrete type when cloned. This scenario
keeps both exception templates in persistent storage and borrows no exception beyond its task cycle.
</description>
*)

{attribute 'no_explicit_call' := 'do not call this function block directly'}
FUNCTION_BLOCK DiagnosticProbe EXTENDS TOF_Testing.SingleCycleTest
VAR_INPUT
	ThrowNative : BOOL;
	ThrowOnGetMessage : BOOL;
END_VAR
VAR_OUTPUT
	BodyCalls : UDINT;
	TeardownCalls : UDINT;
END_VAR
VAR
	_Exception : TOF_Core.StandardException;
	_FormattingFailure : ThrowingGetMessageException;
	_LongMessage : TOF_Core.ERROR_MESSAGE;
END_VAR
VAR_STAT
	//! <summary>Class name shared by all instances of this function block.</summary>
	{attribute 'hide'}
	_ClassName : STRING := __POUNAME();
END_VAR
VAR
	{attribute 'hide'}
	{attribute 'init_namespace'}
	_NamespaceName : STRING;
END_VAR

(*!
<summary>Clears per-run observations.</summary>
*)
METHOD PROTECTED BeforeTest
BodyCalls := 0;
TeardownCalls := 0;
END_METHOD

(*!
<summary>Raises one selected error after recording one body invocation.</summary>
*)
METHOD PROTECTED ExecuteTest
VAR
	i : UDINT;
END_VAR
BodyCalls := BodyCalls + 1;

IF ThrowNative THEN
	Tc2_System.F_RaiseException(ExceptionCode := __SYSTEM.ExceptionCode.RTSEXCPT_ARRAYBOUNDS);
ELSIF ThrowOnGetMessage THEN
	_FormattingFailure.Throw(
		sourceNamespaceName := NamespaceName,
		sourceClassName := ClassName,
		sourcePOUName := __POUNAME(),
		sourcePosition := __POSITION(),
		message := "Original exception with a failing formatter"
	);
ELSE
	_LongMessage := "Long diagnostic: ";

	FOR i := 1 TO 400 DO
		TOF_Core.WideStrings.AppendFit(targetString := _LongMessage, sourceString := "x");
	END_FOR

	TOF_Core.WideStrings.AppendFit(targetString := _LongMessage, sourceString := " END_OF_LONG_DIAGNOSTIC");
	_Exception.Throw(
		sourceNamespaceName := NamespaceName,
		sourceClassName := ClassName,
		sourcePOUName := __POUNAME(),
		sourcePosition := __POSITION(),
		message := _LongMessage
	);
END_IF
END_METHOD

(*!
<summary>Records one cleanup after the captured error.</summary>
*)
METHOD PROTECTED AfterTest
TeardownCalls := TeardownCalls + 1;
END_METHOD

//! <summary>Borrows the concrete class name for the lifetime of this instance; callers must not modify it.</summary>
{attribute 'monitoring' := 'call'}
PROPERTY ClassName : REFERENCE TO STRING
GET
ClassName REF= _ClassName;
END_GET
END_PROPERTY

//! <summary>Borrows the compiler-initialized namespace; callers must not modify the returned reference.</summary>
{attribute 'monitoring' := 'call'}
PROPERTY NamespaceName : REFERENCE TO STRING
GET
NamespaceName REF= _NamespaceName;
END_GET
END_PROPERTY

//! <summary>Reports the complete concrete instance size, excluding separately allocated storage.</summary>
{attribute 'monitoring' := 'call'}
PROPERTY SelfSize : ULINT
GET
SelfSize := XSIZEOF(THIS^);
END_GET
END_PROPERTY

END_FUNCTION_BLOCK

// ---- Tests/Tasks/QueueCleanup/ThrowingGetMessageException.TcPOU
(*
SPDX-FileCopyrightText: © 2026 Oleksandr Tiutyk <trofimich@gmail.com>
SPDX-License-Identifier: MIT
License: https://opensource.org/license/mit
*)

(*!
<summary>Provides a test exception whose GetMessage deliberately throws another exception.</summary>
<description>
Static Throw clones this concrete type. The clone is task-managed; GetMessage deliberately throws a separate
StandardException. The per-instance call count records formatter invocations and is independent of diagnostic
payload. This fixture never performs I/O or throws from lifecycle initialization.
</description>
*)

{attribute 'enable_dynamic_creation'}
FUNCTION_BLOCK ThrowingGetMessageException EXTENDS TOF_Core.StandardException
VAR
	_FixtureClassName : STRING := __POUNAME();
	_MessageReadCount : UDINT;
END_VAR

{attribute 'monitoring' := 'call'}
PROPERTY ClassName : REFERENCE TO STRING
GET
ClassName REF= _FixtureClassName;
END_GET
END_PROPERTY

(*!
<summary>Creates a task-managed clone retaining the failing formatter.</summary>
<description>
Registers the new object before copying inherited diagnostics. Its formatter invocation count starts at zero.
The caller borrows the result until task cleanup. Allocation failure follows the framework terminal policy.
</description>
*)
METHOD Clone : TOF_Core.IObject
VAR
	copy : POINTER TO ThrowingGetMessageException;
END_VAR
copy := __NEW(ThrowingGetMessageException);

IF copy = 0 THEN
	TOF_Core.DynamicMemoryManager.RaiseAllocationFailure();
END_IF

TOF_Core.DynamicMemoryManager.RegisterAutoDisposedObject(autoDisposedObject := copy^);
copy^.CopyGeneralFields(sourceException := THIS^);
Clone := copy^;
END_METHOD

(*!
<summary>Deliberately fails while formatting the original child exception.</summary>
<description>
Counts the call before throwing so tests can distinguish formatter failure from early refusal.
Neither formatting option is used.
</description>
<param name="showSource">Unused formatting option retained for the inherited signature.</param>
<param name="timestampDisplayMode">Unused formatting option retained for the inherited signature.</param>
*)
METHOD GetMessage : TOF_Core.ERROR_MESSAGE
VAR_INPUT
	showSource : BOOL := FALSE;
	timestampDisplayMode : TOF_Core.TIMESTAMP_DISPLAY_MODE := TOF_Core.TIMESTAMP_DISPLAY_MODE.HIDDEN;
END_VAR
VAR
	failure : TOF_Core.StandardException;
END_VAR
_MessageReadCount := _MessageReadCount + 1;

failure.Throw(
	sourceNamespaceName := NamespaceName,
	sourceClassName := ClassName,
	sourcePOUName := __POUNAME(),
	sourcePosition := __POSITION(),
	message := "Injected message formatting failure"
);
END_METHOD

(*!
<summary>Borrows the test library namespace.</summary>
*)

{attribute 'monitoring' := 'call'}
PROPERTY NamespaceName : REFERENCE TO STRING
GET
NamespaceName REF= CurrentNamespace.Name;
END_GET
END_PROPERTY

(*!
<summary>Reports the concrete fixture size.</summary>
*)

{attribute 'monitoring' := 'call'}
PROPERTY SelfSize : ULINT
GET
SelfSize := XSIZEOF(THIS^);
END_GET
END_PROPERTY

//! <summary>Counts this instance's formatter calls, including ones that raised the injected exception.</summary>
PROPERTY MessageReadCount : UDINT
GET
MessageReadCount := _MessageReadCount;
END_GET
END_PROPERTY

END_FUNCTION_BLOCK

// ---- Tests/Testing/AssertionTestRunner.TcPOU
(*
SPDX-License-Identifier: MIT
License: https://opensource.org/license/mit
*)

(*!
<summary>Runs the twenty-seven independent assertion contract scenarios.</summary>
<description>
Owns persistent root instances and fixed child storage. Use from one task without reentry.
Children borrows the same array for the instance lifetime. Root parents remain zero.
</description>
*)

{attribute 'no_assign'}
{attribute 'no_explicit_call' := 'do not call this function block directly'}
FUNCTION_BLOCK AssertionTestRunner EXTENDS TOF_Testing.TestRunner<27>
VAR_STAT
	//! <summary>Class name shared by instances of this concrete runner.</summary>
	{attribute 'hide'}
	_ClassName : STRING := __POUNAME();
END_VAR
VAR
	{attribute 'hide'}
	{attribute 'init_namespace'}
	_NamespaceName : STRING;
END_VAR
VAR_OUTPUT
	//! <summary>Owned root element used by this runner.</summary>
	Assertion0 : AssertionContractProbe(name := "FLOAT_TOLERANCE", parent := 0);
	//! <summary>Owned root element used by this runner.</summary>
	Assertion1 : AssertionContractProbe(name := "INTEGER_EXACT", parent := 0);
	//! <summary>Owned root element used by this runner.</summary>
	Assertion2 : AssertionContractProbe(name := "TYPED_LITERALS", parent := 0);
	//! <summary>Owned root element used by this runner.</summary>
	Assertion3 : AssertionContractProbe(name := "MESSAGE_CHAIN", parent := 0);
	//! <summary>Owned root element used by this runner.</summary>
	Assertion4 : AssertionContractProbe(name := "NEGATIVE_TOLERANCE", parent := 0);
	//! <summary>Owned root element used by this runner.</summary>
	Assertion5 : AssertionContractProbe(name := "NAN_TOLERANCE", parent := 0);
	//! <summary>Owned root element used by this runner.</summary>
	Assertion6 : AssertionContractProbe(name := "INFINITE_TOLERANCE", parent := 0);
	//! <summary>Owned root element used by this runner.</summary>
	Assertion7 : AssertionContractProbe(name := "MESSAGE_RESET", parent := 0);
	//! <summary>Owned root element used by this runner.</summary>
	Assertion8 : AssertionContractProbe(name := "POINTERS_AND_STRINGS", parent := 0);
	//! <summary>Owned root element used by this runner.</summary>
	Assertion9 : AssertionContractProbe(name := "FIRST_FAILURE", parent := 0);
	//! <summary>Owned root element used by this runner.</summary>
	Assertion10 : AssertionContractProbe(name := "SPECIAL_FLOATS", parent := 0);
	//! <summary>Owned root element used by this runner.</summary>
	Assertion11 : AssertionContractProbe(name := "OPPOSITE_LIMITS", parent := 0);
	//! <summary>Owned root element used by this runner.</summary>
	Assertion12 : AssertionContractProbe(name := "GENERIC_MESSAGE_CHAIN", parent := 0);
	//! <summary>Owned root element used by this runner.</summary>
	Assertion13 : AssertionContractProbe(name := "GENERIC_MESSAGE_RESET", parent := 0);
	//! <summary>Owned independent-context regression scenario.</summary>
	Assertion14 : AssertionContractProbe(name := "CONTEXT_TRANSITIONS", parent := 0);
	//! <summary>Owned independent-context regression scenario.</summary>
	Assertion15 : AssertionContractProbe(name := "TYPED_MESSAGE_AFTER_GENERIC", parent := 0);
	//! <summary>Owned independent-context regression scenario.</summary>
	Assertion16 : AssertionContractProbe(name := "GENERIC_MESSAGE_AFTER_TYPED", parent := 0);
	//! <summary>Owned independent-context regression scenario.</summary>
	Assertion17 : AssertionContractProbe(name := "TYPED_MESSAGE_RESET_AFTER_GENERIC", parent := 0);
	//! <summary>Owned independent-context regression scenario.</summary>
	Assertion18 : AssertionContractProbe(name := "INTEGER_FAILURE", parent := 0);
	//! <summary>Owned independent-context regression scenario.</summary>
	Assertion19 : AssertionContractProbe(name := "BITSTRING_FAILURE", parent := 0);
	//! <summary>Owned independent-context regression scenario.</summary>
	Assertion20 : AssertionContractProbe(name := "POINTER_FAILURE", parent := 0);
	//! <summary>Owned independent-context regression scenario.</summary>
	Assertion21 : AssertionContractProbe(name := "STRING_LONG_FAILURE", parent := 0);
	//! <summary>Owned independent-context regression scenario.</summary>
	Assertion22 : AssertionContractProbe(name := "WIDE_STRING_LONG_FAILURE", parent := 0);
	//! <summary>Owned independent-context regression scenario.</summary>
	Assertion23 : AssertionContractProbe(name := "STRING_CONTAINMENT_FAILURE", parent := 0);
	//! <summary>Owned independent-context regression scenario.</summary>
	Assertion24 : AssertionContractProbe(name := "FLOAT_ORDERING_FAILURE", parent := 0);
	//! <summary>Owned independent-context regression scenario.</summary>
	Assertion25 : AssertionContractProbe(name := "FLOAT_EQUALITY_FAILURE", parent := 0);
	//! <summary>Owned independent-context regression scenario.</summary>
	Assertion26 : AssertionContractProbe(name := "TIME_ORDERING_FAILURE", parent := 0);
END_VAR
VAR
	_Children : ARRAY [0.._ChildCount - 1] OF TOF_Testing.ITestElement :=
	[
		Assertion0,
		Assertion1,
		Assertion2,
		Assertion3,
		Assertion4,
		Assertion5,
		Assertion6,
		Assertion7,
		Assertion8,
		Assertion9,
		Assertion10,
		Assertion11,
		Assertion12,
		Assertion13,
		Assertion14,
		Assertion15,
		Assertion16,
		Assertion17,
		Assertion18,
		Assertion19,
		Assertion20,
		Assertion21,
		Assertion22,
		Assertion23,
		Assertion24,
		Assertion25,
		Assertion26
	];
END_VAR

(*!
<summary>Borrows the concrete class name; callers must not modify the returned storage.</summary>
*)
{attribute 'monitoring' := 'call'}
PROPERTY ClassName : REFERENCE TO STRING
GET
ClassName REF= _ClassName;
END_GET
END_PROPERTY

(*!
<summary>Borrows the concrete namespace name for the instance lifetime; callers must not modify it.</summary>
*)
{attribute 'monitoring' := 'call'}
PROPERTY NamespaceName : REFERENCE TO STRING
GET
NamespaceName REF= _NamespaceName;
END_GET
END_PROPERTY

(*!
<summary>Reports the complete concrete instance size.</summary>
*)
{attribute 'monitoring' := 'call'}
PROPERTY SelfSize : ULINT
GET
SelfSize := XSIZEOF(THIS^);
END_GET
END_PROPERTY

(*!
<summary>Borrows the unchanged persistent root array; application code must not modify it.</summary>
*)
{attribute 'monitoring' := 'call'}
PROPERTY Children : REFERENCE TO ARRAY [0.._ChildCount - 1] OF TOF_Testing.ITestElement
GET
Children REF= _Children;
END_GET
END_PROPERTY

END_FUNCTION_BLOCK

// ---- Tests/Testing/AssertionContractProbe.TcPOU
(*
SPDX-FileCopyrightText: © 2026 Oleksandr Tiutyk <trofimich@gmail.com>
SPDX-License-Identifier: MIT
License: https://opensource.org/license/mit
*)

(*!
<summary>Exercises typed literal assertions, borrowed values and chain-wide diagnostics.</summary>
<description>
Each persistent instance runs one selected scenario. Expected failures are checked by the independent runner contract suite.
Raw NaN construction avoids arithmetic that could raise before the assertion begins.
Independent-context scenarios cover type transitions, native predicates and failed typed diagnostics.
</description>
*)

{attribute 'no_explicit_call' := 'do not call this function block directly'}
FUNCTION_BLOCK AssertionContractProbe EXTENDS TOF_Testing.SingleCycleTest
VAR_INPUT
	Scenario : ASSERTION_PROBE_SCENARIO;
END_VAR
VAR
	_Exception : TOF_Core.StandardException;
END_VAR
VAR_STAT
	//! <summary>Class name shared by all instances of this function block.</summary>
	{attribute 'hide'}
	_ClassName : STRING := __POUNAME();
END_VAR
VAR
	{attribute 'hide'}
	{attribute 'init_namespace'}
	_NamespaceName : STRING;
END_VAR

(*!
<summary>Verifies that a later teardown exception cannot replace the first assertion failure.</summary>
*)
METHOD PROTECTED AfterTest
IF Scenario = ASSERTION_PROBE_SCENARIO.FIRST_FAILURE THEN
	_Exception.Throw(
		sourceNamespaceName := NamespaceName,
		sourceClassName := ClassName,
		sourcePOUName := __POUNAME(),
		sourcePosition := __POSITION(),
		message := "Later teardown diagnostic"
	);
END_IF
END_METHOD

//! <summary>Borrows the concrete class name for the lifetime of this instance; callers must not modify it.</summary>
{attribute 'monitoring' := 'call'}
PROPERTY ClassName : REFERENCE TO STRING
GET
ClassName REF= _ClassName;
END_GET
END_PROPERTY

(*!
<summary>Checks both Core bit results and exact assertion equality for a pair of floating encodings.</summary>
<description>
Both inputs must represent the same canonical value. The expected binary64 encoding is an independent test vector.
</description>
<param name="realBits">Stored binary32 operand.</param>
<param name="longRealBits">Stored binary64 operand.</param>
<param name="expectedBits">Expected canonical binary64 result for both operands.</param>
*)
METHOD PRIVATE checkCanonicalPair
VAR_INPUT
	realBits : UDINT;
	longRealBits : ULINT;
	expectedBits : ULINT;
END_VAR
VAR
	narrow : TOF_Core.REAL_UNION;
	wide : TOF_Core.LREAL_UNION;
	expected : TOF_Core.LREAL_UNION;
END_VAR
narrow.Raw := realBits;
wide.Raw := longRealBits;
expected.Raw := expectedBits;

Assert.ThatULInt(actual := TOF_Core.Reals.GetCanonicalBinary64Bits(value := narrow.Value)).ToBe(expected := expectedBits);
Assert.ThatULInt(actual := TOF_Core.LongReals.GetCanonicalBinary64Bits(value := wide.Value)).ToBe(expected := expectedBits);

Assert.That(actual := narrow.Value).ToBe(expected := wide.Value);
Assert.ThatLongReal(actual := wide.Value).ToBe(expected := expected.Value);
END_METHOD

